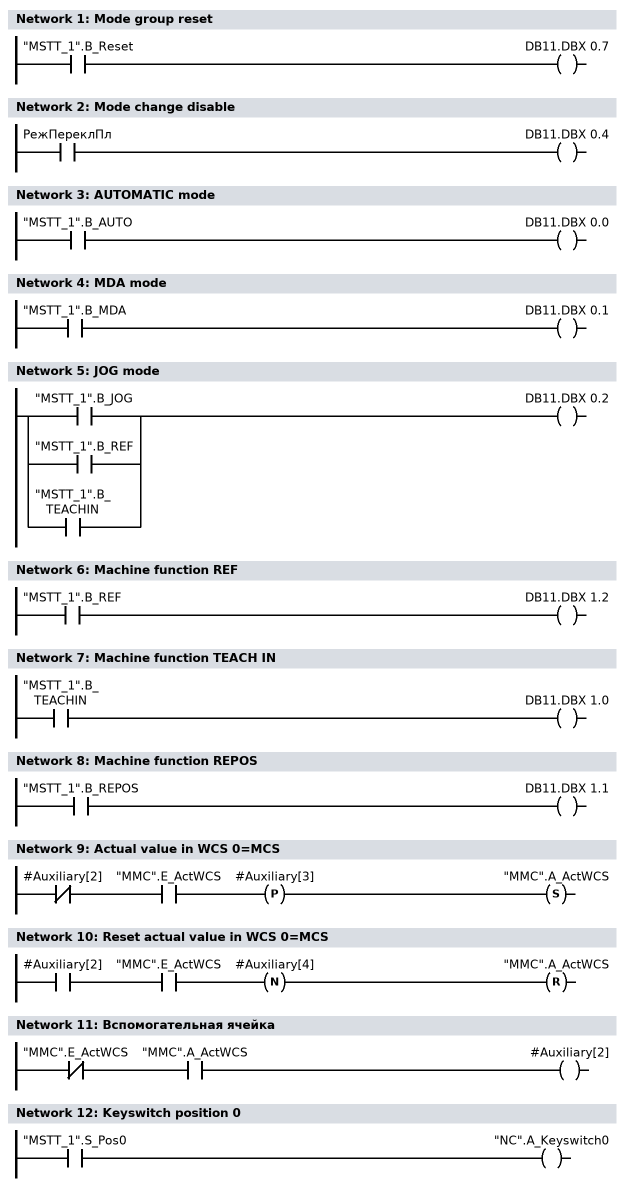
[picture p24: Lathe_Modes networks 1-12]
NETWORK
TITLE = Mode group reset
      A     "MSTT_1".B_Reset;
      =     DB11.DBX 0.7;
NETWORK
TITLE = Mode change disable 
      A     "РежПереклПл";
      =     DB11.DBX 0.4;
NETWORK
TITLE = AUTOMATIC mode
      A     "MSTT_1".B_AUTO;
      =     DB11.DBX 0.0;
NETWORK
TITLE = MDA mode
      A     "MSTT_1".B_MDA;
      =     DB11.DBX 0.1;
NETWORK
TITLE = JOG mode
      O     "MSTT_1".B_JOG;
      O     "MSTT_1".B_REF;
      O     "MSTT_1".B_TEACHIN;
      =     DB11.DBX 0.2;
NETWORK
TITLE = Machine function REF
      A     "MSTT_1".B_REF;
      =     DB11.DBX 1.2;
NETWORK
TITLE = Machine function TEACH IN
      A     "MSTT_1".B_TEACHIN;
      =     DB11.DBX 1.0;
NETWORK
TITLE = Machine function REPOS
      A     "MSTT_1".B_REPOS;
      =     DB11.DBX 1.1;
NETWORK
TITLE = Actual value in WCS 0=MCS
      AN    #Auxiliary[2];
      A     "MMC".E_ActWCS;
      FP    #Auxiliary[3];
      S     "MMC".A_ActWCS;
NETWORK
TITLE = Reset actual value in WCS 0=MCS
      A     #Auxiliary[2];
      A     "MMC".E_ActWCS;
      FN    #Auxiliary[4];
      R     "MMC".A_ActWCS;
NETWORK
TITLE = Вспомогательная ячейка
      AN    "MMC".E_ActWCS;
      A     "MMC".A_ActWCS;
      =     #Auxiliary[2];
NETWORK
TITLE = Keyswitch position 0
      A     "MSTT_1".S_Pos0;
      =     "NC".A_Keyswitch0;
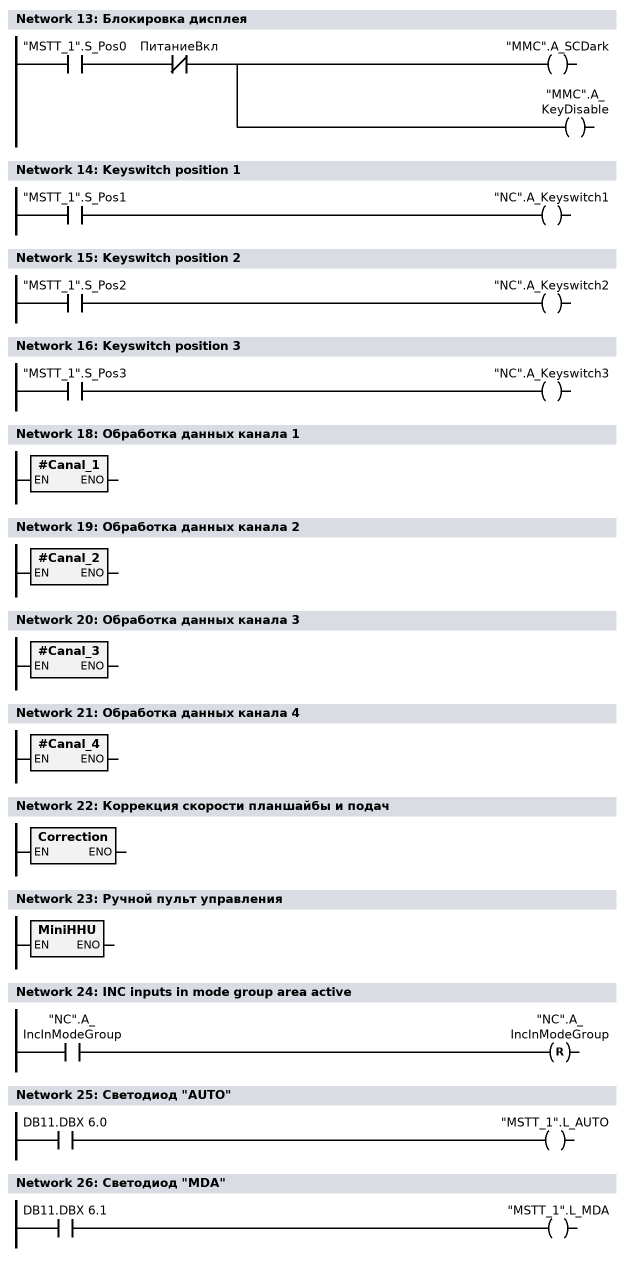
NETWORK
TITLE = Блокировка дисплея
      A     "MSTT_1".S_Pos0;
      AN    "ПитаниеВкл";
      =     "MMC".A_SCDark;
      =     "MMC".A_KeyDisable;
NETWORK
TITLE = Keyswitch position 1
      A     "MSTT_1".S_Pos1;
      =     "NC".A_Keyswitch1;
NETWORK
TITLE = Keyswitch position 2
      A     "MSTT_1".S_Pos2;
      =     "NC".A_Keyswitch2;
NETWORK
TITLE = Keyswitch position 3
      A     "MSTT_1".S_Pos3;
      =     "NC".A_Keyswitch3;
NETWORK
TITLE = Обработка вспомогательных функций
//      CALL  FC   107
      NOP   0;
NETWORK
TITLE = Обработка данных канала 1
      CALL  #Canal_1;
      NOP   0;
NETWORK
TITLE = Обработка данных канала 2
      CALL  #Canal_2;
      NOP   0;
NETWORK
TITLE = Обработка данных канала 3
      CALL  #Canal_3;
      NOP   0;
NETWORK
TITLE = Обработка данных канала 4
      CALL  #Canal_4;
      NOP   0;
NETWORK
TITLE = Коррекция скорости планшайбы и подач
      CALL  "Correction";
      NOP   0;
NETWORK
TITLE = Ручной пульт управления
      CALL  "MiniHHU";
      NOP   0;
NETWORK
TITLE = INC inputs in mode group area active
      A     "NC".A_IncInModeGroup;
      R     "NC".A_IncInModeGroup;
NETWORK
TITLE = Светодиод "AUTO"
      A     DB11.DBX 6.0;
      =     "MSTT_1".L_AUTO;
NETWORK
TITLE = Светодиод "MDA"
      A     DB11.DBX 6.1;
      =     "MSTT_1".L_MDA;
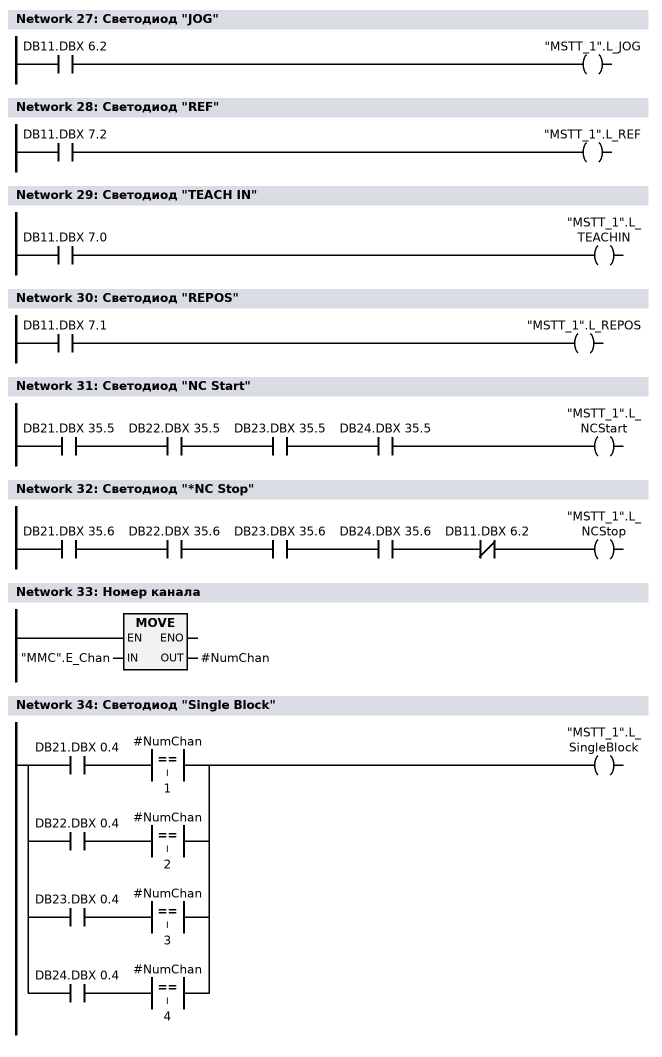
NETWORK
TITLE = Светодиод "JOG"
      A     DB11.DBX 6.2;
      =     "MSTT_1".L_JOG;
NETWORK
TITLE = Светодиод "REF"
      A     DB11.DBX 7.2;
      =     "MSTT_1".L_REF;
NETWORK
TITLE = Светодиод "TEACH IN"
      A     DB11.DBX 7.0;
      =     "MSTT_1".L_TEACHIN;
NETWORK
TITLE = Светодиод "REPOS"
      A     DB11.DBX 7.1;
      =     "MSTT_1".L_REPOS;
NETWORK
TITLE = Светодиод "NC Start"
      A     DB21.DBX 35.5;
      A     DB22.DBX 35.5;
      A     DB23.DBX 35.5;
      A     DB24.DBX 35.5;
      =     "MSTT_1".L_NCStart;
NETWORK
TITLE = Светодиод "*NC Stop"
      A     DB21.DBX 35.6;
      A     DB22.DBX 35.6;
      A     DB23.DBX 35.6;
      A     DB24.DBX 35.6;
      AN    DB11.DBX 6.2;
      =     "MSTT_1".L_NCStop;
NETWORK
TITLE = Номер канала
      L     "MMC".E_Chan;
      T     #NumChan;
      NOP   0;
NETWORK
TITLE = Светодиод "Single Block"
      A     DB21.DBX 0.4;
      A(;
      L     #NumChan;
      L     1;
      ==I;
      );
      O;
      A     DB22.DBX 0.4;
      A(;
      L     #NumChan;
      L     2;
      ==I;
      );
      O;
      A     DB23.DBX 0.4;
      A(;
      L     #NumChan;
      L     3;
      ==I;
      );
      O;
      A     DB24.DBX 0.4;
      A(;
      L     #NumChan;
      L     4;
      ==I;
      );
      =     "MSTT_1".L_SingleBlock;
END_FUNCTION_BLOCK

FUNCTION_BLOCK "Channel1_Modes"	// FB 106
AUTHOR : SEDIN
VERSION : 0.1
VAR
  Auxiliary : ARRAY  [0 .. 15 ] OF //Вспомогательная ячейка
  BOOL ;
  Table : FB 100;
  Support : FB 101;
END_VAR
VAR_TEMP
  NumChan : INT ;	//Номер канала
  B_SingleBlock : BOOL ;	//Клавиша SingleBlock
END_VAR
BEGIN
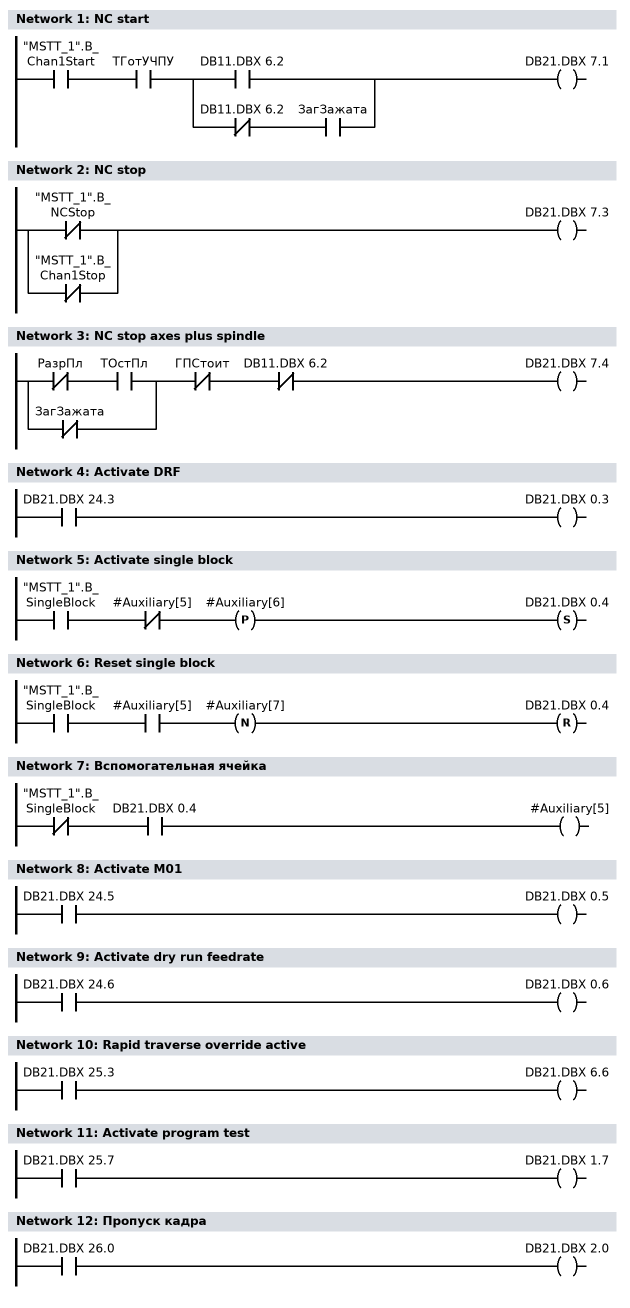
NETWORK
TITLE = NC start
      A     "MSTT_1".B_Chan1Start;
      A     "ТГотУЧПУ";
      A(;
      O     DB11.DBX 6.2;
      O;
      AN    DB11.DBX 6.2;
      A     "ЗагЗажата";
      );
      =     DB21.DBX 7.1;
NETWORK
TITLE = NC stop
      ON    "MSTT_1".B_NCStop;
      ON    "MSTT_1".B_Chan1Stop;
      =     DB21.DBX 7.3;
NETWORK
TITLE = NC stop axes plus spindle
      A(;
      AN    "РазрПл";
      A     "ТОстПл";
      ON    "ЗагЗажата";
      );
      AN    "ГПСтоит";
      AN    DB11.DBX 6.2;
      =     DB21.DBX 7.4;
NETWORK
TITLE = Activate DRF
      A     DB21.DBX 24.3;
      =     DB21.DBX 0.3;
NETWORK
TITLE = Activate single block
      A     "MSTT_1".B_SingleBlock;
      AN    #Auxiliary[5];
      FP    #Auxiliary[6];
      S     DB21.DBX 0.4;
NETWORK
TITLE = Reset single block
      A     "MSTT_1".B_SingleBlock;
      A     #Auxiliary[5];
      FN    #Auxiliary[7];
      R     DB21.DBX 0.4;
NETWORK
TITLE = Вспомогательная ячейка
      AN    "MSTT_1".B_SingleBlock;
      A     DB21.DBX 0.4;
      =     #Auxiliary[5];
NETWORK
TITLE = Activate M01
      A     DB21.DBX 24.5;
      =     DB21.DBX 0.5;
NETWORK
TITLE = Activate dry run feedrate
      A     DB21.DBX 24.6;
      =     DB21.DBX 0.6;
NETWORK
TITLE = Rapid traverse override active
      A     DB21.DBX 25.3;
      =     DB21.DBX 6.6;
NETWORK
TITLE = Activate program test
      A     DB21.DBX 25.7;
      =     DB21.DBX 1.7;
NETWORK
TITLE = Пропуск кадра
      A     DB21.DBX 26.0;
      =     DB21.DBX 2.0;
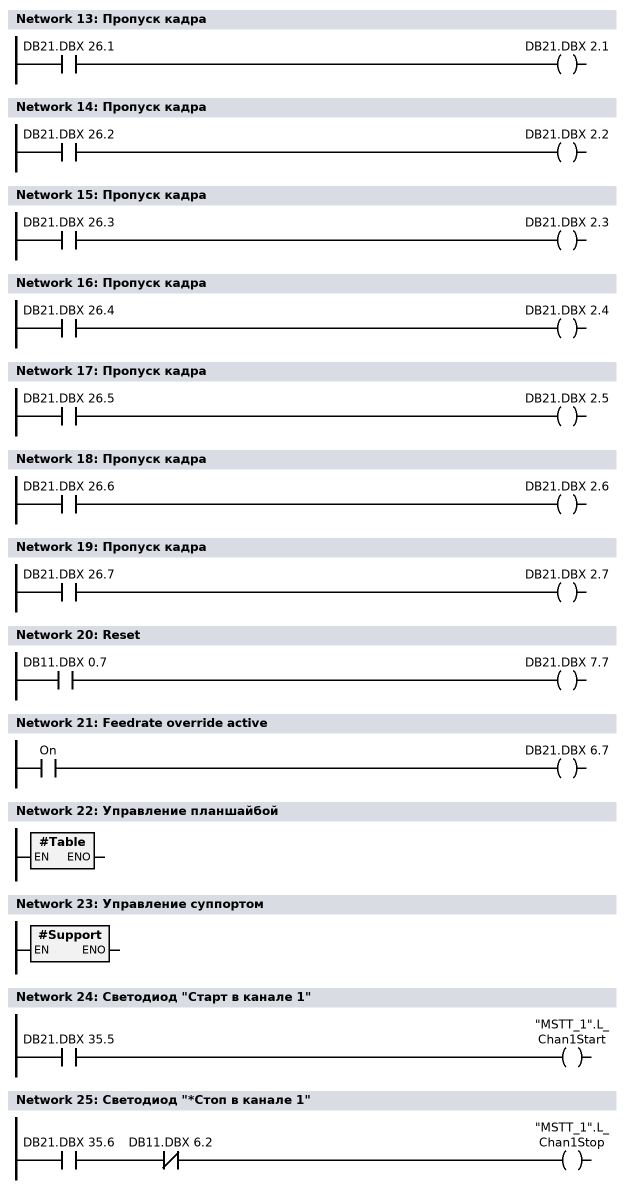
NETWORK
TITLE = Пропуск кадра
      A     DB21.DBX 26.1;
      =     DB21.DBX 2.1;
NETWORK
TITLE = Пропуск кадра
      A     DB21.DBX 26.2;
      =     DB21.DBX 2.2;
NETWORK
TITLE = Пропуск кадра
      A     DB21.DBX 26.3;
      =     DB21.DBX 2.3;
NETWORK
TITLE = Пропуск кадра
      A     DB21.DBX 26.4;
      =     DB21.DBX 2.4;
NETWORK
TITLE = Пропуск кадра
      A     DB21.DBX 26.5;
      =     DB21.DBX 2.5;
NETWORK
TITLE = Пропуск кадра
      A     DB21.DBX 26.6;
      =     DB21.DBX 2.6;
NETWORK
TITLE = Пропуск кадра
      A     DB21.DBX 26.7;
      =     DB21.DBX 2.7;
NETWORK
TITLE = Reset
      A     DB11.DBX 0.7;
      =     DB21.DBX 7.7;
NETWORK
TITLE = Feedrate override active
      A     "On";
      =     DB21.DBX 6.7;
NETWORK
TITLE = Управление планшайбой
      CALL  #Table;
      NOP   0;
NETWORK
TITLE = Управление суппортом
      CALL  #Support;
      NOP   0;
NETWORK
TITLE = Светодиод "Старт в канале 1"
      A     DB21.DBX 35.5;
      =     "MSTT_1".L_Chan1Start;
NETWORK
TITLE = Светодиод "*Стоп в канале 1"
      A     DB21.DBX 35.6;
      AN    DB11.DBX 6.2;
      =     "MSTT_1".L_Chan1Stop;
END_FUNCTION_BLOCK

FUNCTION_BLOCK "Channel2_Modes"	// FB 107
AUTHOR : SEDIN
VERSION : 0.1
VAR
  Auxiliary : ARRAY  [0 .. 15 ] OF //Вспомогательная ячейка
  BOOL ;
  Support : FB 102;
END_VAR
VAR_TEMP
  NumChan : INT ;	//Номер канала
  B_SingleBlock : BOOL ;	//Клавиша SingleBlock
END_VAR
BEGIN
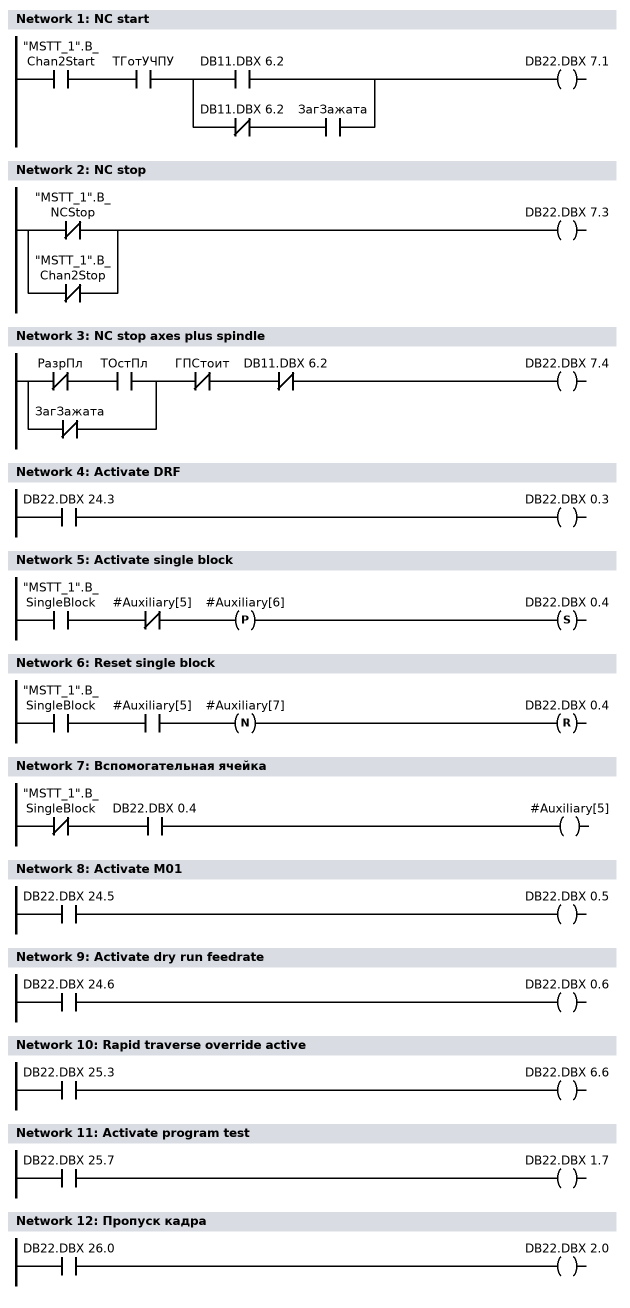
NETWORK
TITLE = NC start
      A     "MSTT_1".B_Chan2Start;
      A     "ТГотУЧПУ";
      A(;
      O     DB11.DBX 6.2;
      O;
      AN    DB11.DBX 6.2;
      A     "ЗагЗажата";
      );
      =     DB22.DBX 7.1;
NETWORK
TITLE = NC stop
      ON    "MSTT_1".B_NCStop;
      ON    "MSTT_1".B_Chan2Stop;
      =     DB22.DBX 7.3;
NETWORK
TITLE = NC stop axes plus spindle
      A(;
      AN    "РазрПл";
      A     "ТОстПл";
      ON    "ЗагЗажата";
      );
      AN    "ГПСтоит";
      AN    DB11.DBX 6.2;
      =     DB22.DBX 7.4;
NETWORK
TITLE = Activate DRF
      A     DB22.DBX 24.3;
      =     DB22.DBX 0.3;
NETWORK
TITLE = Activate single block
      A     "MSTT_1".B_SingleBlock;
      AN    #Auxiliary[5];
      FP    #Auxiliary[6];
      S     DB22.DBX 0.4;
NETWORK
TITLE = Reset single block
      A     "MSTT_1".B_SingleBlock;
      A     #Auxiliary[5];
      FN    #Auxiliary[7];
      R     DB22.DBX 0.4;
NETWORK
TITLE = Вспомогательная ячейка
      AN    "MSTT_1".B_SingleBlock;
      A     DB22.DBX 0.4;
      =     #Auxiliary[5];
NETWORK
TITLE = Activate M01
      A     DB22.DBX 24.5;
      =     DB22.DBX 0.5;
NETWORK
TITLE = Activate dry run feedrate
      A     DB22.DBX 24.6;
      =     DB22.DBX 0.6;
NETWORK
TITLE = Rapid traverse override active
      A     DB22.DBX 25.3;
      =     DB22.DBX 6.6;
NETWORK
TITLE = Activate program test
      A     DB22.DBX 25.7;
      =     DB22.DBX 1.7;
NETWORK
TITLE = Пропуск кадра
      A     DB22.DBX 26.0;
      =     DB22.DBX 2.0;
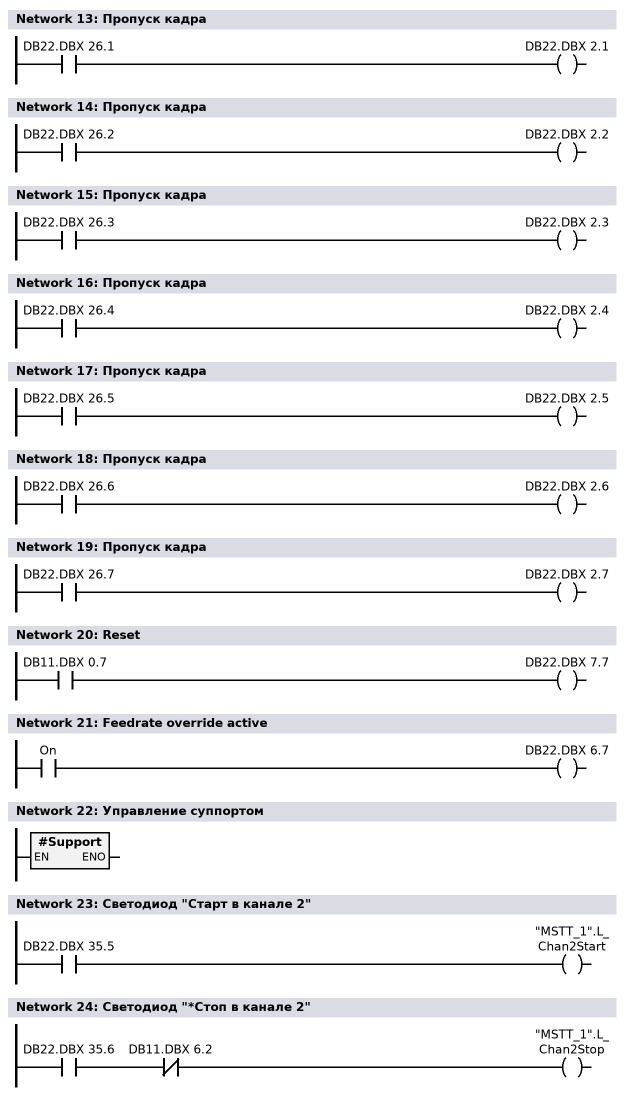
NETWORK
TITLE = Пропуск кадра
      A     DB22.DBX 26.1;
      =     DB22.DBX 2.1;
NETWORK
TITLE = Пропуск кадра
      A     DB22.DBX 26.2;
      =     DB22.DBX 2.2;
NETWORK
TITLE = Пропуск кадра
      A     DB22.DBX 26.3;
      =     DB22.DBX 2.3;
NETWORK
TITLE = Пропуск кадра
      A     DB22.DBX 26.4;
      =     DB22.DBX 2.4;
NETWORK
TITLE = Пропуск кадра
      A     DB22.DBX 26.5;
      =     DB22.DBX 2.5;
NETWORK
TITLE = Пропуск кадра
      A     DB22.DBX 26.6;
      =     DB22.DBX 2.6;
NETWORK
TITLE = Пропуск кадра
      A     DB22.DBX 26.7;
      =     DB22.DBX 2.7;
NETWORK
TITLE = Reset
      A     DB11.DBX 0.7;
      =     DB22.DBX 7.7;
NETWORK
TITLE = Feedrate override active
      A     "On";
      =     DB22.DBX 6.7;
NETWORK
TITLE = Управление суппортом
      CALL  #Support;
      NOP   0;
NETWORK
TITLE = Светодиод "Старт в канале 2"
      A     DB22.DBX 35.5;
      =     "MSTT_1".L_Chan2Start;
NETWORK
TITLE = Светодиод "*Стоп в канале 2"
      A     DB22.DBX 35.6;
      AN    DB11.DBX 6.2;
      =     "MSTT_1".L_Chan2Stop;
END_FUNCTION_BLOCK

FUNCTION_BLOCK "Channel3_Modes"	// FB 108
AUTHOR : SEDIN
VERSION : 0.1
VAR
  Auxiliary : ARRAY  [0 .. 15 ] OF //Вспомогательная ячейка
  BOOL ;
  Support : FB 103;
END_VAR
VAR_TEMP
  NumChan : INT ;	//Номер канала
  B_SingleBlock : BOOL ;	//Клавиша SingleBlock
END_VAR
BEGIN
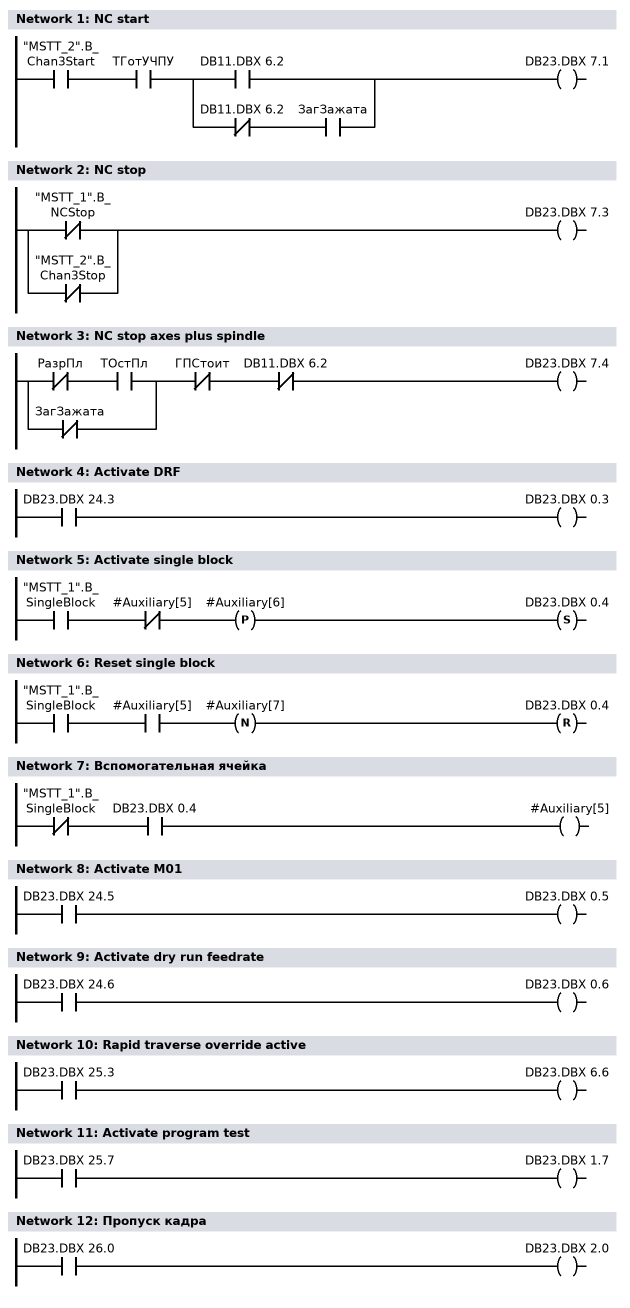
NETWORK
TITLE = NC start
      A     "MSTT_2".B_Chan3Start;
      A     "ТГотУЧПУ";
      A(;
      O     DB11.DBX 6.2;
      O;
      AN    DB11.DBX 6.2;
      A     "ЗагЗажата";
      );
      =     DB23.DBX 7.1;
NETWORK
TITLE = NC stop
      ON    "MSTT_1".B_NCStop;
      ON    "MSTT_2".B_Chan3Stop;
      =     DB23.DBX 7.3;
NETWORK
TITLE = NC stop axes plus spindle
      A(;
      AN    "РазрПл";
      A     "ТОстПл";
      ON    "ЗагЗажата";
      );
      AN    "ГПСтоит";
      AN    DB11.DBX 6.2;
      =     DB23.DBX 7.4;
NETWORK
TITLE = Activate DRF
      A     DB23.DBX 24.3;
      =     DB23.DBX 0.3;
NETWORK
TITLE = Activate single block
      A     "MSTT_1".B_SingleBlock;
      AN    #Auxiliary[5];
      FP    #Auxiliary[6];
      S     DB23.DBX 0.4;
NETWORK
TITLE = Reset single block
      A     "MSTT_1".B_SingleBlock;
      A     #Auxiliary[5];
      FN    #Auxiliary[7];
      R     DB23.DBX 0.4;
NETWORK
TITLE = Вспомогательная ячейка
      AN    "MSTT_1".B_SingleBlock;
      A     DB23.DBX 0.4;
      =     #Auxiliary[5];
NETWORK
TITLE = Activate M01
      A     DB23.DBX 24.5;
      =     DB23.DBX 0.5;
NETWORK
TITLE = Activate dry run feedrate
      A     DB23.DBX 24.6;
      =     DB23.DBX 0.6;
NETWORK
TITLE = Rapid traverse override active
      A     DB23.DBX 25.3;
      =     DB23.DBX 6.6;
NETWORK
TITLE = Activate program test
      A     DB23.DBX 25.7;
      =     DB23.DBX 1.7;
NETWORK
TITLE = Пропуск кадра
      A     DB23.DBX 26.0;
      =     DB23.DBX 2.0;
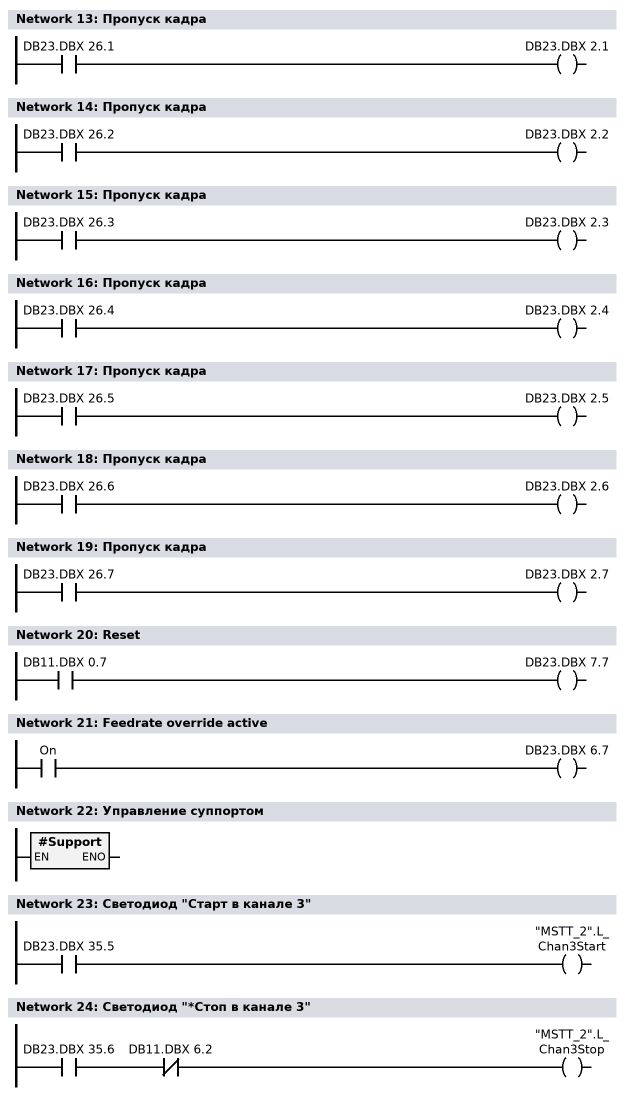
NETWORK
TITLE = Пропуск кадра
      A     DB23.DBX 26.1;
      =     DB23.DBX 2.1;
NETWORK
TITLE = Пропуск кадра
      A     DB23.DBX 26.2;
      =     DB23.DBX 2.2;
NETWORK
TITLE = Пропуск кадра
      A     DB23.DBX 26.3;
      =     DB23.DBX 2.3;
NETWORK
TITLE = Пропуск кадра
      A     DB23.DBX 26.4;
      =     DB23.DBX 2.4;
NETWORK
TITLE = Пропуск кадра
      A     DB23.DBX 26.5;
      =     DB23.DBX 2.5;
NETWORK
TITLE = Пропуск кадра
      A     DB23.DBX 26.6;
      =     DB23.DBX 2.6;
NETWORK
TITLE = Пропуск кадра
      A     DB23.DBX 26.7;
      =     DB23.DBX 2.7;
NETWORK
TITLE = Reset
      A     DB11.DBX 0.7;
      =     DB23.DBX 7.7;
NETWORK
TITLE = Feedrate override active
      A     "On";
      =     DB23.DBX 6.7;
NETWORK
TITLE = Управление суппортом
      CALL  #Support;
      NOP   0;
NETWORK
TITLE = Светодиод "Старт в канале 3"
      A     DB23.DBX 35.5;
      =     "MSTT_2".L_Chan3Start;
NETWORK
TITLE = Светодиод "*Стоп в канале 3"
      A     DB23.DBX 35.6;
      AN    DB11.DBX 6.2;
      =     "MSTT_2".L_Chan3Stop;
END_FUNCTION_BLOCK

FUNCTION_BLOCK "Channel4_Modes"	// FB 109
AUTHOR : SEDIN
VERSION : 0.1
VAR
  Auxiliary : ARRAY  [0 .. 15 ] OF //Вспомогательная ячейка
  BOOL ;
  Support : FB 104;
END_VAR
VAR_TEMP
  NumChan : INT ;	//Номер канала
  B_SingleBlock : BOOL ;	//Клавиша SingleBlock
END_VAR
BEGIN
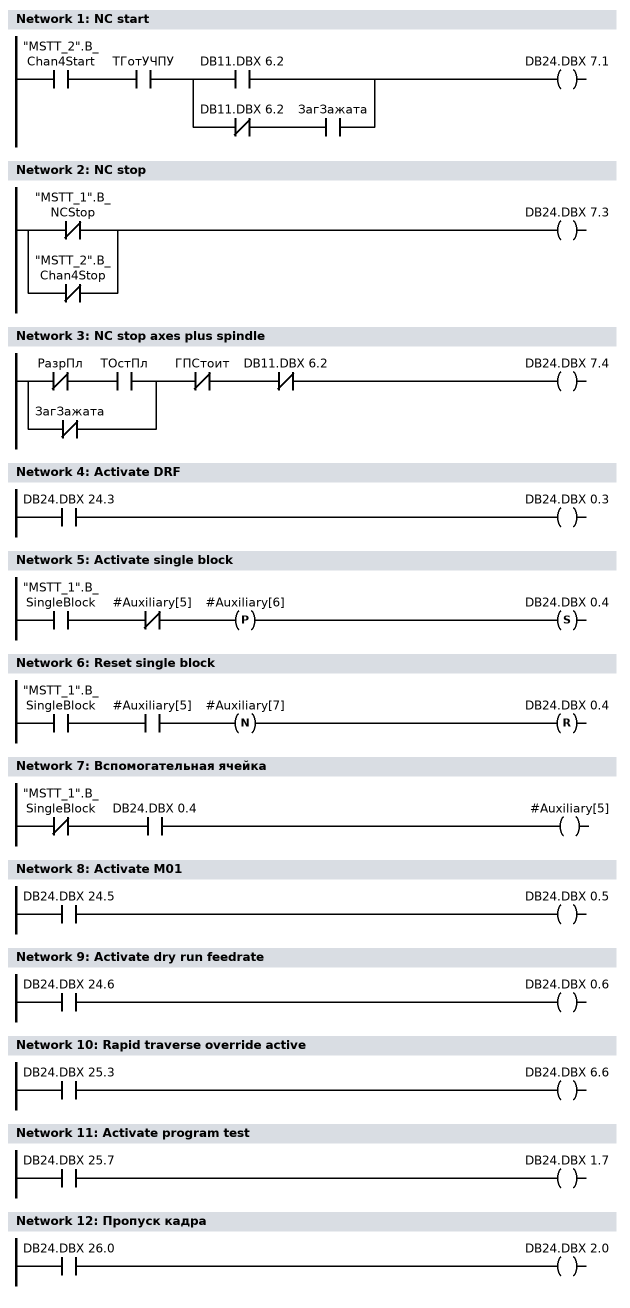
NETWORK
TITLE = NC start
      A     "MSTT_2".B_Chan4Start;
      A     "ТГотУЧПУ";
      A(;
      O     DB11.DBX 6.2;
      O;
      AN    DB11.DBX 6.2;
      A     "ЗагЗажата";
      );
      =     DB24.DBX 7.1;
NETWORK
TITLE = NC stop
      ON    "MSTT_1".B_NCStop;
      ON    "MSTT_2".B_Chan4Stop;
      =     DB24.DBX 7.3;
NETWORK
TITLE = NC stop axes plus spindle
      A(;
      AN    "РазрПл";
      A     "ТОстПл";
      ON    "ЗагЗажата";
      );
      AN    "ГПСтоит";
      AN    DB11.DBX 6.2;
      =     DB24.DBX 7.4;
NETWORK
TITLE = Activate DRF
      A     DB24.DBX 24.3;
      =     DB24.DBX 0.3;
NETWORK
TITLE = Activate single block
      A     "MSTT_1".B_SingleBlock;
      AN    #Auxiliary[5];
      FP    #Auxiliary[6];
      S     DB24.DBX 0.4;
NETWORK
TITLE = Reset single block
      A     "MSTT_1".B_SingleBlock;
      A     #Auxiliary[5];
      FN    #Auxiliary[7];
      R     DB24.DBX 0.4;
NETWORK
TITLE = Вспомогательная ячейка
      AN    "MSTT_1".B_SingleBlock;
      A     DB24.DBX 0.4;
      =     #Auxiliary[5];
NETWORK
TITLE = Activate M01
      A     DB24.DBX 24.5;
      =     DB24.DBX 0.5;
NETWORK
TITLE = Activate dry run feedrate
      A     DB24.DBX 24.6;
      =     DB24.DBX 0.6;
NETWORK
TITLE = Rapid traverse override active
      A     DB24.DBX 25.3;
      =     DB24.DBX 6.6;
NETWORK
TITLE = Activate program test
      A     DB24.DBX 25.7;
      =     DB24.DBX 1.7;
NETWORK
TITLE = Пропуск кадра
      A     DB24.DBX 26.0;
      =     DB24.DBX 2.0;
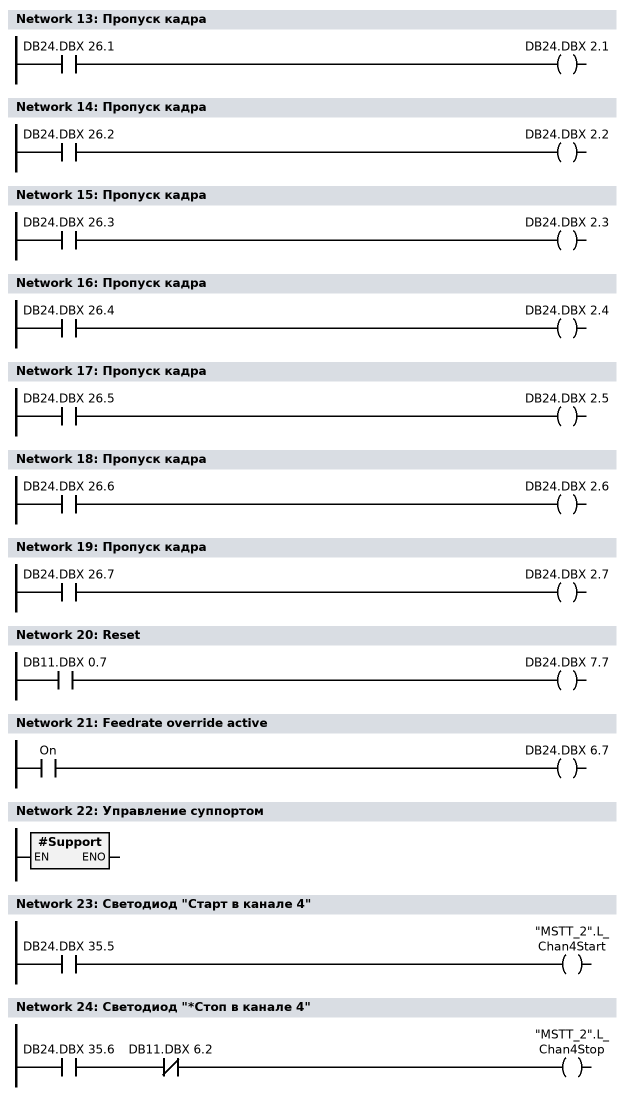
NETWORK
TITLE = Пропуск кадра
      A     DB24.DBX 26.1;
      =     DB24.DBX 2.1;
NETWORK
TITLE = Пропуск кадра
      A     DB24.DBX 26.2;
      =     DB24.DBX 2.2;
NETWORK
TITLE = Пропуск кадра
      A     DB24.DBX 26.3;
      =     DB24.DBX 2.3;
NETWORK
TITLE = Пропуск кадра
      A     DB24.DBX 26.4;
      =     DB24.DBX 2.4;
NETWORK
TITLE = Пропуск кадра
      A     DB24.DBX 26.5;
      =     DB24.DBX 2.5;
NETWORK
TITLE = Пропуск кадра
      A     DB24.DBX 26.6;
      =     DB24.DBX 2.6;
NETWORK
TITLE = Пропуск кадра
      A     DB24.DBX 26.7;
      =     DB24.DBX 2.7;
NETWORK
TITLE = Reset
      A     DB11.DBX 0.7;
      =     DB24.DBX 7.7;
NETWORK
TITLE = Feedrate override active
      A     "On";
      =     DB24.DBX 6.7;
NETWORK
TITLE = Управление суппортом
      CALL  #Support;
      NOP   0;
NETWORK
TITLE = Светодиод "Старт в канале 4"
      A     DB24.DBX 35.5;
      =     "MSTT_2".L_Chan4Start;
NETWORK
TITLE = Светодиод "*Стоп в канале 4"
      A     DB24.DBX 35.6;
      AN    DB11.DBX 6.2;
      =     "MSTT_2".L_Chan4Stop;
END_FUNCTION_BLOCK

FUNCTION_BLOCK "Support_Lub"	// FB 121
AUTHOR : SEDIN
VERSION : 0.1
VAR_INPUT
  Permission : BOOL ;	//Разрешение работы насоса ИСС
  LubButton : BOOL ;	//Кнопка принудительной прокачки ИСС
  Pressure : BOOL ;	//Реле давления ИСС
  Level : BOOL ;	//Реле уровня ИСС
  BlockError : BOOL ;	//Блокировка ошибки смазки
END_VAR
VAR_OUTPUT
  Pump : BOOL ;	//Команда на смазку суппорта
  LubError : BOOL ;	//Ошибка смазки суппорта
  Message1 : BOOL ;	//Сообщение о низком уровне масла
  Message2 : BOOL ;	//Сообщение об отсутствии набора давления
  Message3 : BOOL ;	//Сообщение об отсутствии падения давления
END_VAR
VAR
  Mem_1 : BOOL ;	//Память фронта сигнала 1
  Mem_2 : BOOL ;	//Память фронта сигнала 2
  ResetTimers : BOOL ;	//Сброс таймеров смазки суппорта
  TLubError_In : BOOL ;	//Пуск таймера задержки реакции на ошибку смазки
  TLubInterval_In : BOOL ;	//Пуск таймера интервала прокачки ИСС
  TLubDelay_In : BOOL ;	//Пуск таймера задержки на прокачку ИСС
  TLubError_Q : BOOL ;	//Таймер задержки реакции на ошибку смазки сработал
  TLubInterval_Q : BOOL ;	//Таймер интервала прокачки ИСС сработал
  TLubDelay_Q : BOOL ;	//Таймер задержки на прокачку ИСС сработал
  TLubError : SFB 4;	//Задержка реакции на ошибку смазки
  TLubInterval : SFB 4;	//Таймер интервала прокачки ИСС
  TLubDelay : SFB 4;	//Задержка на прокачку ИСС
END_VAR
BEGIN
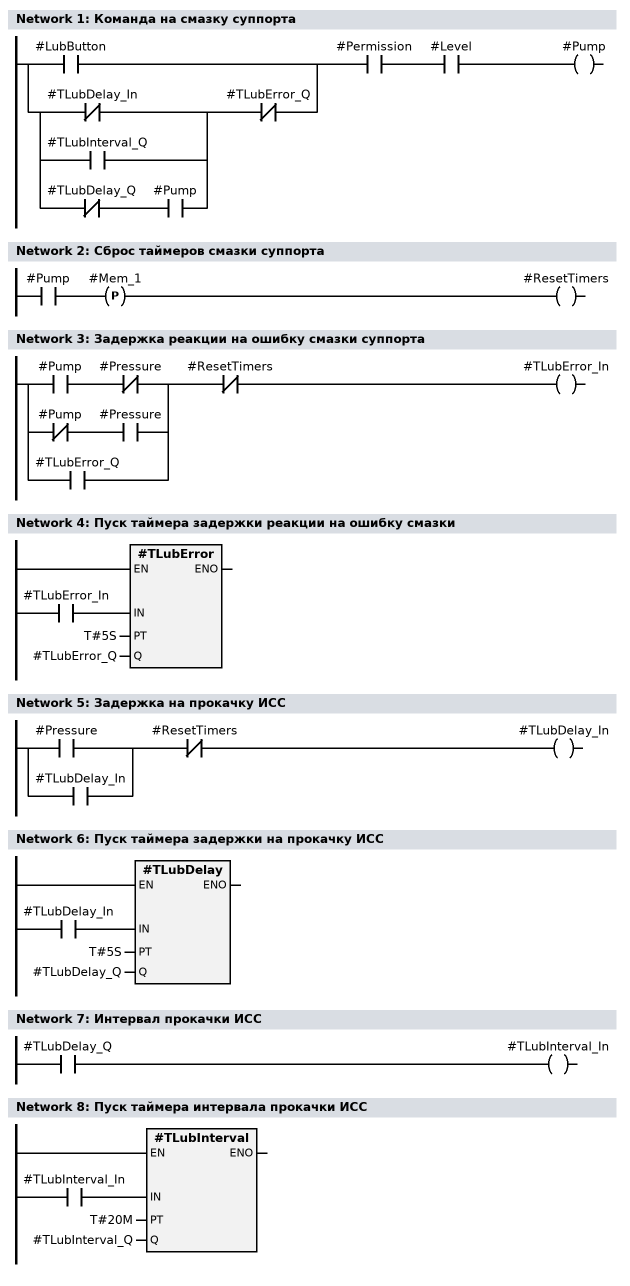
NETWORK
TITLE = Команда на смазку суппорта
      A(;
      O     #LubButton;
      O;
      A(;
      ON    #TLubDelay_In;
      O     #TLubInterval_Q;
      O;
      AN    #TLubDelay_Q;
      A     #Pump;
      );
      AN    #TLubError_Q;
      );
      A     #Permission;
      A     #Level;
      =     #Pump;
NETWORK
TITLE = Сброс таймеров смазки суппорта
      A     #Pump;
      FP    #Mem_1;
      =     #ResetTimers;
NETWORK
TITLE = Задержка реакции на ошибку смазки суппорта
      A(;
      A     #Pump;
      AN    #Pressure;
      O;
      AN    #Pump;
      A     #Pressure;
      O     #TLubError_Q;
      );
      AN    #ResetTimers;
      =     #TLubError_In;
NETWORK
TITLE = Пуск таймера задержки реакции на ошибку смазки
      A     #TLubError_In;
      =     L 0.0;
      BLD   103;
      CALL  #TLubError (
           IN                       := L 0.0,
           PT                       := T#5S,
           Q                        := #TLubError_Q);
      NOP   0;
NETWORK
TITLE = Задержка на прокачку ИСС
      A(;
      O     #Pressure;
      O     #TLubDelay_In;
      );
      AN    #ResetTimers;
      =     #TLubDelay_In;
NETWORK
TITLE = Пуск таймера задержки на прокачку ИСС 
      A     #TLubDelay_In;
      =     L 0.0;
      BLD   103;
      CALL  #TLubDelay (
           IN                       := L 0.0,
           PT                       := T#5S,
           Q                        := #TLubDelay_Q);
      NOP   0;
NETWORK
TITLE = Интервал прокачки ИСС
      A     #TLubDelay_Q;
      =     #TLubInterval_In;
NETWORK
TITLE = Пуск таймера интервала прокачки ИСС
      A     #TLubInterval_In;
      =     L 0.0;
      BLD   103;
      CALL  #TLubInterval (
           IN                       := L 0.0,
           PT                       := T#20M,
           Q                        := #TLubInterval_Q);
      NOP   0;
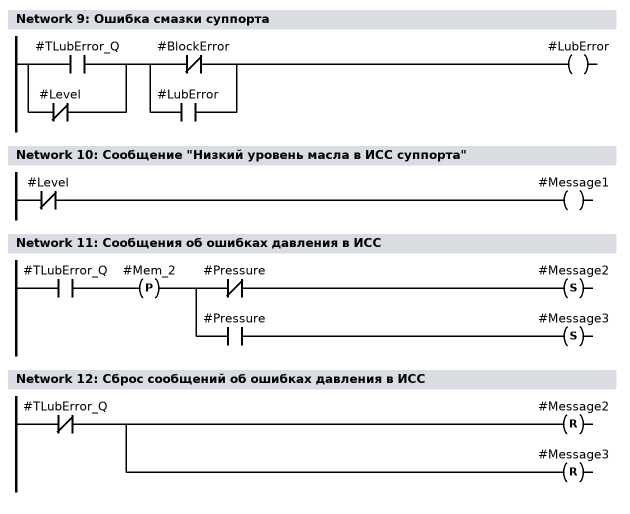
NETWORK
TITLE = Ошибка смазки суппорта
      A(;
      O     #TLubError_Q;
      ON    #Level;
      );
      A(;
      ON    #BlockError;
      O     #LubError;
      );
      =     #LubError;
NETWORK
TITLE = Сообщение "Низкий уровень масла в ИСС суппорта"
      AN    #Level;
      =     #Message1;
NETWORK
TITLE = Сообщения об ошибках давления в ИСС
      A     #TLubError_Q;
      FP    #Mem_2;
      =     L 0.0;
      A     L 0.0;
      AN    #Pressure;
      S     #Message2;
      A     L 0.0;
      A     #Pressure;
      S     #Message3;
NETWORK
TITLE = Сброс сообщений об ошибках давления в ИСС
      AN    #TLubError_Q;
      R     #Message2;
      R     #Message3;
END_FUNCTION_BLOCK

FUNCTION_BLOCK FB 1001
AUTHOR : SEDIN
VERSION : 0.1
VAR
  Auxiliary : ARRAY  [0 .. 15 ] OF //Вспомогательная ячейка
  BOOL ;
END_VAR
VAR_TEMP
  ActMoment : INT ;	//Текущий момент, ось 1
END_VAR
BEGIN
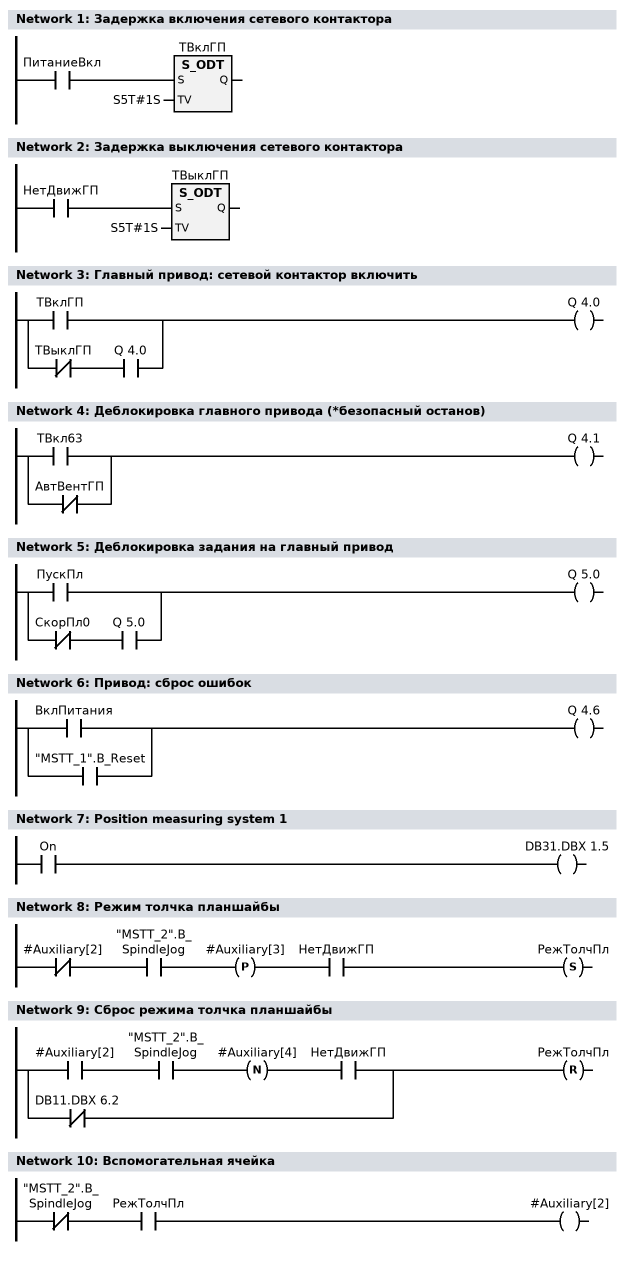
NETWORK
TITLE = Задержка включения сетевого контактора
      A     "ПитаниеВкл";
      L     S5T#1S;
      SD    "ТВклГП";
      NOP   0;
      NOP   0;
      NOP   0;
      NOP   0;
NETWORK
TITLE = Задержка выключения сетевого контактора
      A     "НетДвижГП";
      L     S5T#1S;
      SD    "ТВыклГП";
      NOP   0;
      NOP   0;
      NOP   0;
      NOP   0;
NETWORK
TITLE = Главный привод: сетевой контактор включить
      O     "ТВклГП";
      O;
      AN    "ТВыклГП";
      A     Q 4.0;
      =     Q 4.0;
NETWORK
TITLE = Деблокировка главного привода (*безопасный останов)
      O     "ТВкл63";
      ON    "АвтВентГП";
      =     Q 4.1;
NETWORK
TITLE = Деблокировка задания на главный привод
      O     "ПускПл";
      O;
      AN    "СкорПл0";
      A     Q 5.0;
      =     Q 5.0;
NETWORK
TITLE = Привод: сброс ошибок
      O     "ВклПитания";
      O     "MSTT_1".B_Reset;
      =     Q 4.6;
NETWORK
TITLE = Position measuring system 1
      A     "On";
      =     DB31.DBX 1.5;
NETWORK
TITLE = Режим толчка планшайбы
      AN    #Auxiliary[2];
      A     "MSTT_2".B_SpindleJog;
      FP    #Auxiliary[3];
      A     "НетДвижГП";
      S     "РежТолчПл";
NETWORK
TITLE = Сброс режима толчка планшайбы
      A     #Auxiliary[2];
      A     "MSTT_2".B_SpindleJog;
      FN    #Auxiliary[4];
      A     "НетДвижГП";
      ON    DB11.DBX 6.2;
      R     "РежТолчПл";
NETWORK
TITLE = Вспомогательная ячейка
      AN    "MSTT_2".B_SpindleJog;
      A     "РежТолчПл";
      =     #Auxiliary[2];
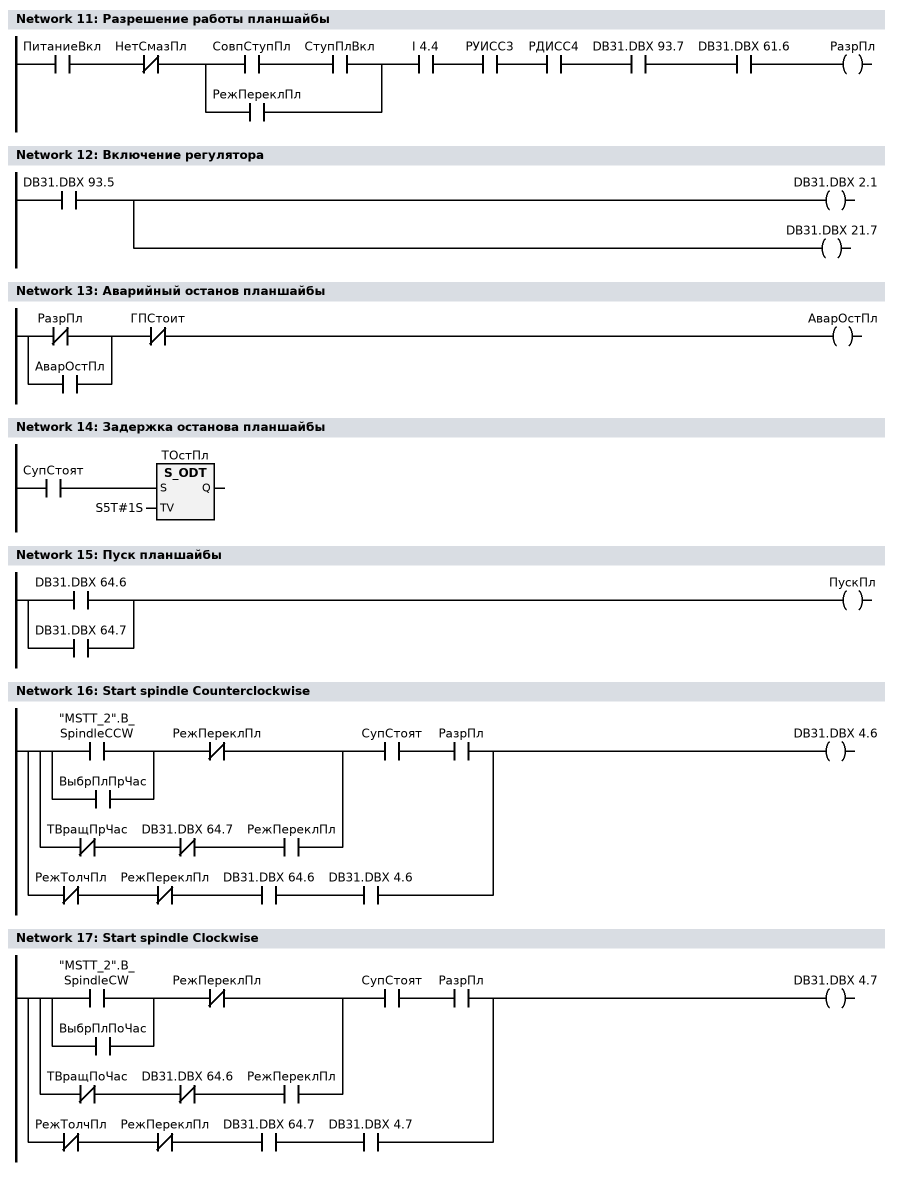
NETWORK
TITLE = Разрешение работы планшайбы
      A     "ПитаниеВкл";
      AN    "НетСмазПл";
      A(;
      A     "СовпСтупПл";
      A     "СтупПлВкл";
      O     "РежПереклПл";
      );
      A     I 4.4;
      A     "РУИСС3";
      A     "РДИСС4";
      A     DB31.DBX 93.7;
      A     DB31.DBX 61.6;
      =     "РазрПл";
NETWORK
TITLE = Включение регулятора
      A     DB31.DBX 93.5;
      =     DB31.DBX 2.1;
      =     DB31.DBX 21.7;
NETWORK
TITLE = Аварийный останов планшайбы
      A(;
      ON    "РазрПл";
      O     "АварОстПл";
      );
      AN    "ГПСтоит";
      =     "АварОстПл";
NETWORK
TITLE = Задержка останова планшайбы
      A     "СупСтоят";
      L     S5T#1S;
      SD    "ТОстПл";
      NOP   0;
      NOP   0;
      NOP   0;
      NOP   0;
NETWORK
TITLE = Пуск планшайбы
      O     DB31.DBX 64.6;
      O     DB31.DBX 64.7;
      =     "ПускПл";
NETWORK
TITLE = Start spindle Counterclockwise
      A(;
      A(;
      O     "MSTT_2".B_SpindleCCW;
      O     "ВыбрПлПрЧас";
      );
      AN    "РежПереклПл";
      O;
      AN    "ТВращПрЧас";
      AN    DB31.DBX 64.7;
      A     "РежПереклПл";
      );
      A     "СупСтоят";
      A     "РазрПл";
      O;
      AN    "РежТолчПл";
      AN    "РежПереклПл";
      A     DB31.DBX 64.6;
      A     DB31.DBX 4.6;
      =     DB31.DBX 4.6;
NETWORK
TITLE = Start spindle Clockwise
      A(;
      A(;
      O     "MSTT_2".B_SpindleCW;
      O     "ВыбрПлПоЧас";
      );
      AN    "РежПереклПл";
      O;
      AN    "ТВращПоЧас";
      AN    DB31.DBX 64.6;
      A     "РежПереклПл";
      );
      A     "СупСтоят";
      A     "РазрПл";
      O;
      AN    "РежТолчПл";
      AN    "РежПереклПл";
      A     DB31.DBX 64.7;
      A     DB31.DBX 4.7;
      =     DB31.DBX 4.7;
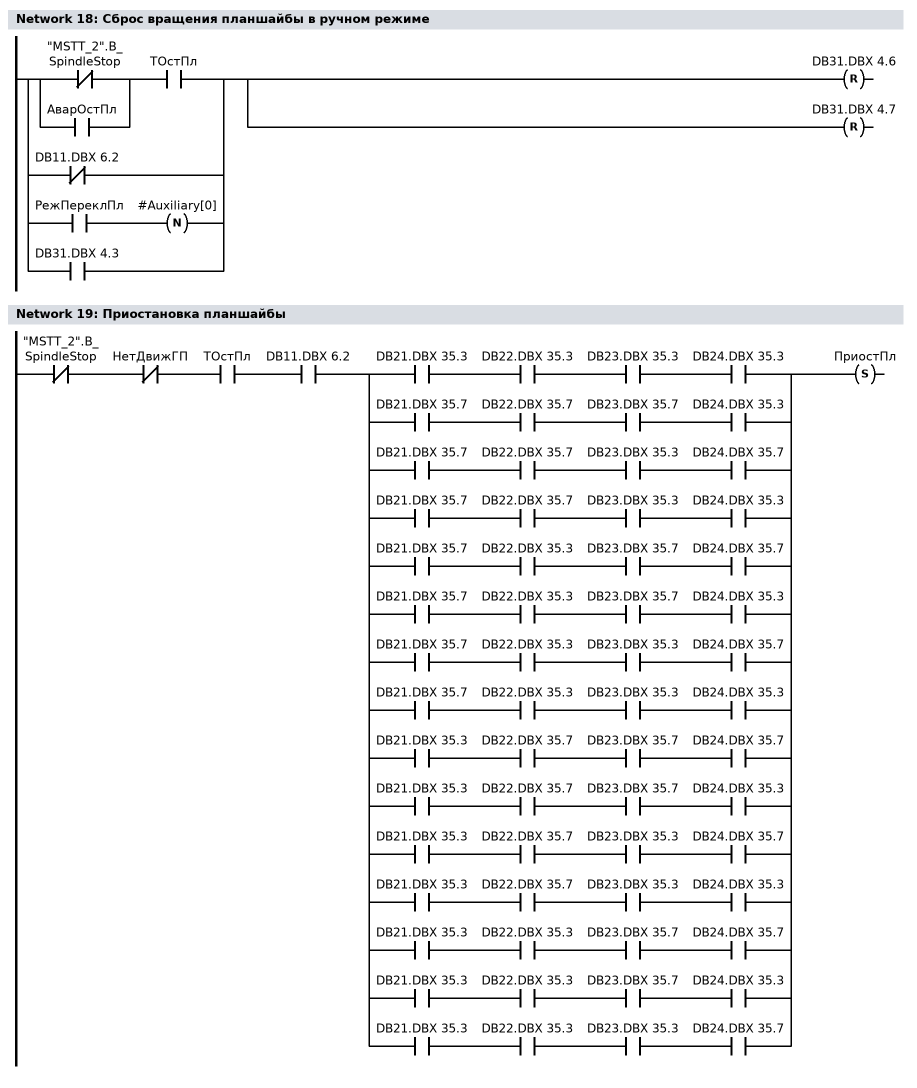
NETWORK
TITLE = Сброс вращения планшайбы в ручном режиме
      A(;
      ON    "MSTT_2".B_SpindleStop;
      O     "АварОстПл";
      );
      A     "ТОстПл";
      ON    DB11.DBX 6.2;
      O(;
      A     "РежПереклПл";
      BLD   100;
      FN    #Auxiliary[0];
      );
      O     DB31.DBX 4.3;
      R     DB31.DBX 4.6;
      R     DB31.DBX 4.7;
NETWORK
TITLE = Приостановка планшайбы
      AN    "MSTT_2".B_SpindleStop;
      AN    "НетДвижГП";
      A     "ТОстПл";
      A     DB11.DBX 6.2;
      A(;
      A     DB21.DBX 35.3;
      A     DB22.DBX 35.3;
      A     DB23.DBX 35.3;
      A     DB24.DBX 35.3;
      O;
      A     DB21.DBX 35.7;
      A     DB22.DBX 35.7;
      A     DB23.DBX 35.7;
      A     DB24.DBX 35.3;
      O;
      A     DB21.DBX 35.7;
      A     DB22.DBX 35.7;
      A     DB23.DBX 35.3;
      A     DB24.DBX 35.7;
      O;
      A     DB21.DBX 35.7;
      A     DB22.DBX 35.7;
      A     DB23.DBX 35.3;
      A     DB24.DBX 35.3;
      O;
      A     DB21.DBX 35.7;
      A     DB22.DBX 35.3;
      A     DB23.DBX 35.7;
      A     DB24.DBX 35.7;
      O;
      A     DB21.DBX 35.7;
      A     DB22.DBX 35.3;
      A     DB23.DBX 35.7;
      A     DB24.DBX 35.3;
      O;
      A     DB21.DBX 35.7;
      A     DB22.DBX 35.3;
      A     DB23.DBX 35.3;
      A     DB24.DBX 35.7;
      O;
      A     DB21.DBX 35.7;
      A     DB22.DBX 35.3;
      A     DB23.DBX 35.3;
      A     DB24.DBX 35.3;
      O;
      A     DB21.DBX 35.3;
      A     DB22.DBX 35.7;
      A     DB23.DBX 35.7;
      A     DB24.DBX 35.7;
      O;
      A     DB21.DBX 35.3;
      A     DB22.DBX 35.7;
      A     DB23.DBX 35.7;
      A     DB24.DBX 35.3;
      O;
      A     DB21.DBX 35.3;
      A     DB22.DBX 35.7;
      A     DB23.DBX 35.3;
      A     DB24.DBX 35.7;
      O;
      A     DB21.DBX 35.3;
      A     DB22.DBX 35.7;
      A     DB23.DBX 35.3;
      A     DB24.DBX 35.3;
      O;
      A     DB21.DBX 35.3;
      A     DB22.DBX 35.3;
      A     DB23.DBX 35.7;
      A     DB24.DBX 35.7;
      O;
      A     DB21.DBX 35.3;
      A     DB22.DBX 35.3;
      A     DB23.DBX 35.7;
      A     DB24.DBX 35.3;
      O;
      A     DB21.DBX 35.3;
      A     DB22.DBX 35.3;
      A     DB23.DBX 35.3;
      A     DB24.DBX 35.7;
      );
      S     "ПриостПл";
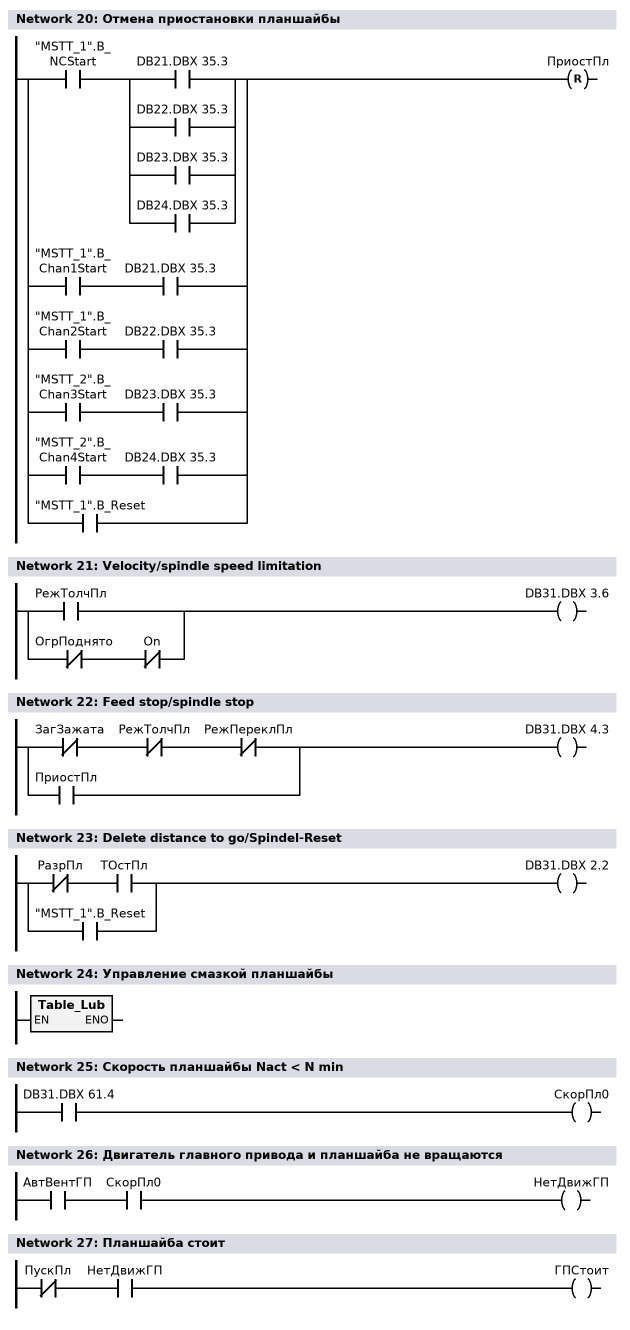
NETWORK
TITLE = Отмена приостановки планшайбы
      A     "MSTT_1".B_NCStart;
      A(;
      O     DB21.DBX 35.3;
      O     DB22.DBX 35.3;
      O     DB23.DBX 35.3;
      O     DB24.DBX 35.3;
      );
      O;
      A     "MSTT_1".B_Chan1Start;
      A     DB21.DBX 35.3;
      O;
      A     "MSTT_1".B_Chan2Start;
      A     DB22.DBX 35.3;
      O;
      A     "MSTT_2".B_Chan3Start;
      A     DB23.DBX 35.3;
      O;
      A     "MSTT_2".B_Chan4Start;
      A     DB24.DBX 35.3;
      O     "MSTT_1".B_Reset;
      R     "ПриостПл";
NETWORK
TITLE = Velocity/spindle speed limitation
      O     "РежТолчПл";
      O;
      AN    "ОгрПоднято";
      AN    "On";
      =     DB31.DBX 3.6;
NETWORK
TITLE = Feed stop/spindle stop
      AN    "ЗагЗажата";
      AN    "РежТолчПл";
      AN    "РежПереклПл";
      O     "ПриостПл";
      =     DB31.DBX 4.3;
NETWORK
TITLE = Delete distance to go/Spindel-Reset
      AN    "РазрПл";
      A     "ТОстПл";
      O     "MSTT_1".B_Reset;
      =     DB31.DBX 2.2;
NETWORK
TITLE = Управление смазкой планшайбы
      CALL  "Table_Lub";
      NOP   0;
NETWORK
TITLE = Скорость планшайбы Nact < N min
      A     DB31.DBX 61.4;
      =     "СкорПл0";
NETWORK
TITLE = Двигатель главного привода и планшайба не вращаются
      A     "АвтВентГП";
      A     "СкорПл0";
      =     "НетДвижГП";
NETWORK
TITLE = Планшайба стоит
      AN    "ПускПл";
      A     "НетДвижГП";
      =     "ГПСтоит";
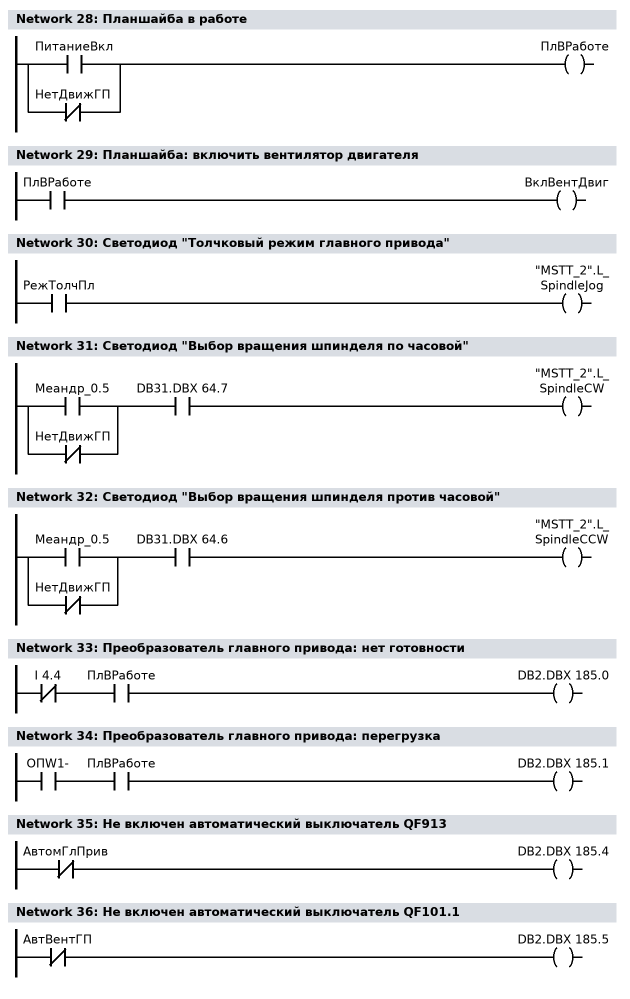
NETWORK
TITLE = Планшайба в работе
      O     "ПитаниеВкл";
      ON    "НетДвижГП";
      =     "ПлВРаботе";
NETWORK
TITLE = Планшайба: включить вентилятор двигателя
      A     "ПлВРаботе";
      =     "ВклВентДвиг";
NETWORK
TITLE = Светодиод "Толчковый режим главного привода"
      A     "РежТолчПл";
      =     "MSTT_2".L_SpindleJog;
NETWORK
TITLE = Светодиод "Выбор вращения шпинделя по часовой"
      A(;
      O     "Меандр_0.5";
      ON    "НетДвижГП";
      );
      A     DB31.DBX 64.7;
      =     "MSTT_2".L_SpindleCW;
NETWORK
TITLE = Светодиод "Выбор вращения шпинделя против часовой"
      A(;
      O     "Меандр_0.5";
      ON    "НетДвижГП";
      );
      A     DB31.DBX 64.6;
      =     "MSTT_2".L_SpindleCCW;
NETWORK
TITLE = Преобразователь главного привода: нет готовности
      AN    I 4.4;
      A     "ПлВРаботе";
      =     DB2.DBX 185.0;
NETWORK
TITLE = Преобразователь главного привода: перегрузка
      A     "ОПW1-";
      A     "ПлВРаботе";
      =     DB2.DBX 185.1;
NETWORK
TITLE = Не включен автоматический выключатель QF913
      AN    "АвтомГлПрив";
      =     DB2.DBX 185.4;
NETWORK
TITLE = Не включен автоматический выключатель QF101.1
      AN    "АвтВентГП";
      =     DB2.DBX 185.5;
END_FUNCTION_BLOCK

// FC 2: know-how protected block, not included

// FC 3: know-how protected block, not included

// FC 5: know-how protected block, not included

// FC 6: know-how protected block, not included

// FC 7: know-how protected block, not included

// FC 8: know-how protected block, not included

// FC 9: know-how protected block, not included

// FC 10: know-how protected block, not included

FUNCTION FC 12 : VOID
AUTHOR : NUMERIK
FAMILY : _800D
NAME : Basics
VERSION : 2.7
VAR_INPUT
  Chan : BYTE ;	//Index of Chan
END_VAR
BEGIN
NETWORK
TITLE =
END_FUNCTION

// FC 13: know-how protected block, not included

// FC 16: know-how protected block, not included

// FC 17: know-how protected block, not included

// FC 18: know-how protected block, not included

// FC 19: know-how protected block, not included

// FC 20: know-how protected block, not included

// FC 21: know-how protected block, not included

// FC 22: know-how protected block, not included

// FC 24: know-how protected block, not included

// FC 25: know-how protected block, not included

// FC 26: know-how protected block, not included

FUNCTION "PowerOn" : VOID	// FC 100
AUTHOR : SEDIN
VERSION : 0.1
VAR_TEMP
  NoMotion : BOOL ;	//Органы станка неподвижны
END_VAR
BEGIN
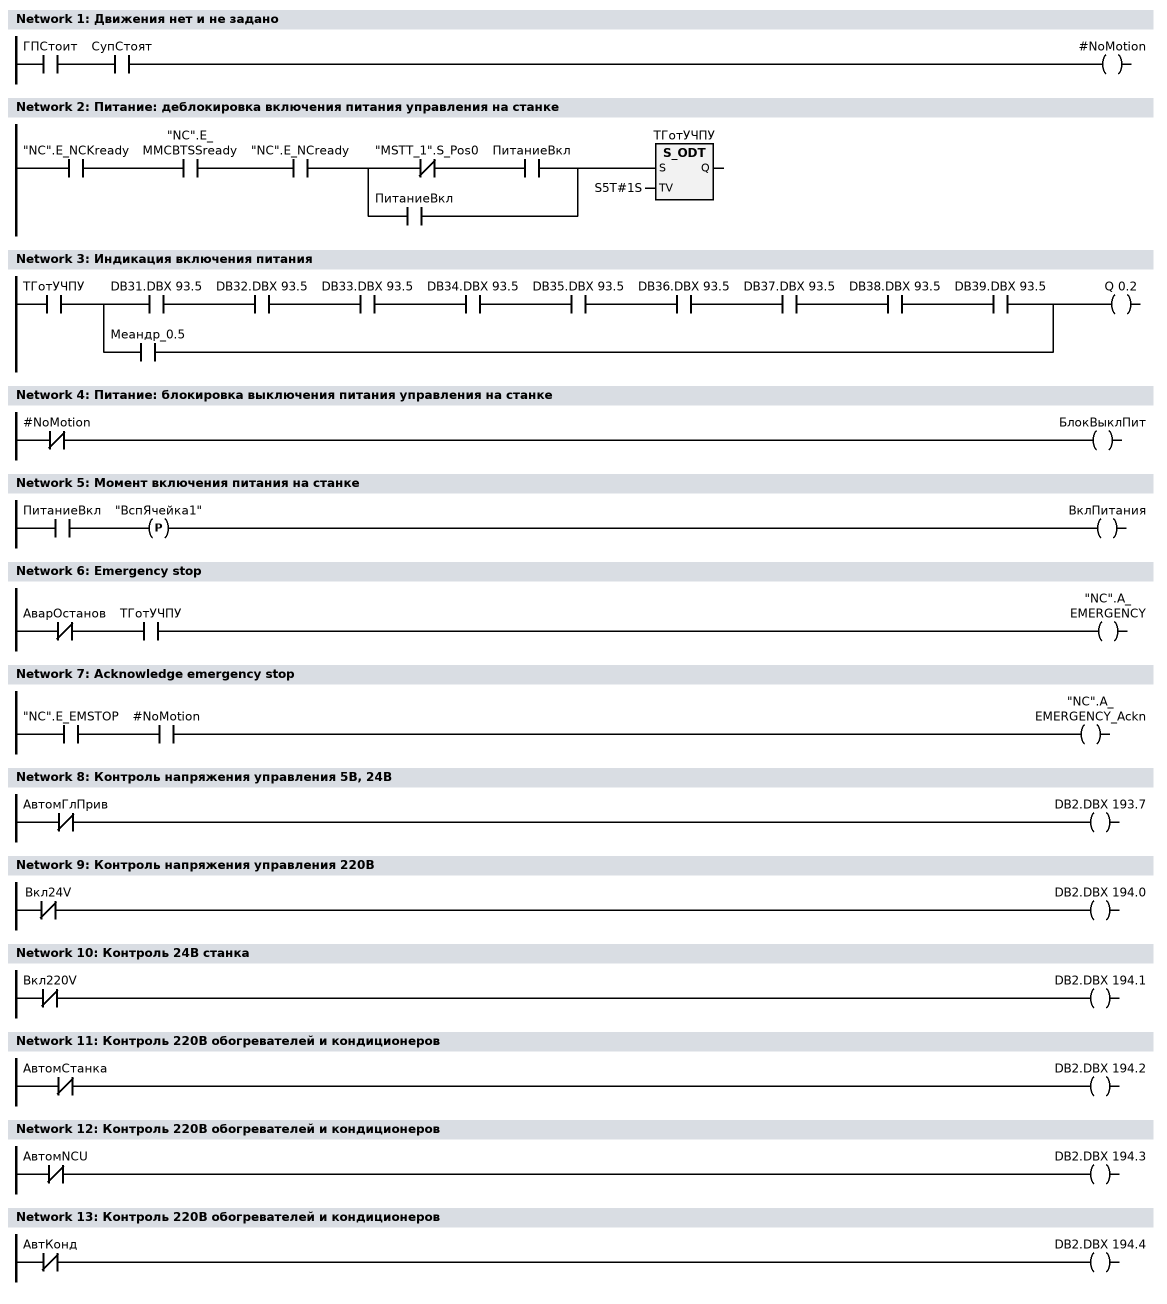
NETWORK
TITLE = Движения нет и не задано
      A     "ГПСтоит";
      A     "СупСтоят";
      =     #NoMotion;
NETWORK
TITLE = Питание: деблокировка включения питания управления на станке
      A     "NC".E_NCKready;
      A     "NC".E_MMCBTSSready;
      A     "NC".E_NCready;
      A(;
      AN    "MSTT_1".S_Pos0;
      A     "ПитаниеВкл";
      O     "ПитаниеВкл";
      );
      L     S5T#1S;
      SD    "ТГотУЧПУ";
      NOP   0;
      NOP   0;
      NOP   0;
      NOP   0;
NETWORK
TITLE = Индикация включения питания
      A     "ТГотУЧПУ";
      A(;
      A     DB31.DBX 93.5;
      A     DB32.DBX 93.5;
      A     DB33.DBX 93.5;
      A     DB34.DBX 93.5;
      A     DB35.DBX 93.5;
      A     DB36.DBX 93.5;
      A     DB37.DBX 93.5;
      A     DB38.DBX 93.5;
      A     DB39.DBX 93.5;
      O     "Меандр_0.5";
      );
      =     Q 0.2;
NETWORK
TITLE = Питание: блокировка выключения питания управления на станке
      AN    #NoMotion;
      =     "БлокВыклПит";
NETWORK
TITLE = Момент включения питания на станке
      A     "ПитаниеВкл";
      BLD   100;
      FP    "ВспЯчейка1";
      =     "ВклПитания";
NETWORK
TITLE = Emergency stop                        
      AN    "АварОстанов";
      A     "ТГотУЧПУ";
      =     "NC".A_EMERGENCY;
NETWORK
TITLE = Acknowledge emergency stop                      
      A     "NC".E_EMSTOP;
      A     #NoMotion;
      =     "NC".A_EMERGENCY_Ackn;
NETWORK
TITLE = Контроль напряжения управления 5В, 24В
      AN    "АвтомГлПрив";
      =     DB2.DBX 193.7;
NETWORK
TITLE = Контроль напряжения управления 220В
      AN    "Вкл24V";
      =     DB2.DBX 194.0;
NETWORK
TITLE = Контроль 24В станка
      AN    "Вкл220V";
      =     DB2.DBX 194.1;
NETWORK
TITLE = Контроль 220В обогревателей и кондиционеров
      AN    "АвтомСтанка";
      =     DB2.DBX 194.2;
NETWORK
TITLE = Контроль 220В обогревателей и кондиционеров
      AN    "АвтомNCU";
      =     DB2.DBX 194.3;
NETWORK
TITLE = Контроль 220В обогревателей и кондиционеров
      AN    "АвтКонд";
      =     DB2.DBX 194.4;
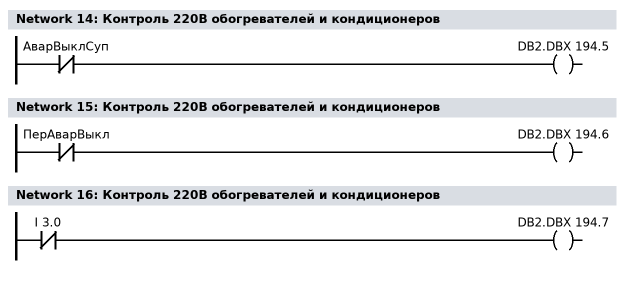
NETWORK
TITLE = Контроль 220В обогревателей и кондиционеров
      AN    "АварВыклСуп";
      =     DB2.DBX 194.5;
NETWORK
TITLE = Контроль 220В обогревателей и кондиционеров
      AN    "ПерАварВыкл";
      =     DB2.DBX 194.6;
NETWORK
TITLE = Контроль 220В обогревателей и кондиционеров
      AN    I 3.0;
      =     DB2.DBX 194.7;
END_FUNCTION

FUNCTION "Infeed_Module" : VOID	// FC 101
AUTHOR : SEDIN
VERSION : 0.1
VAR_TEMP
  Aux : ARRAY  [1 .. 10 ] OF BOOL ;
END_VAR
BEGIN
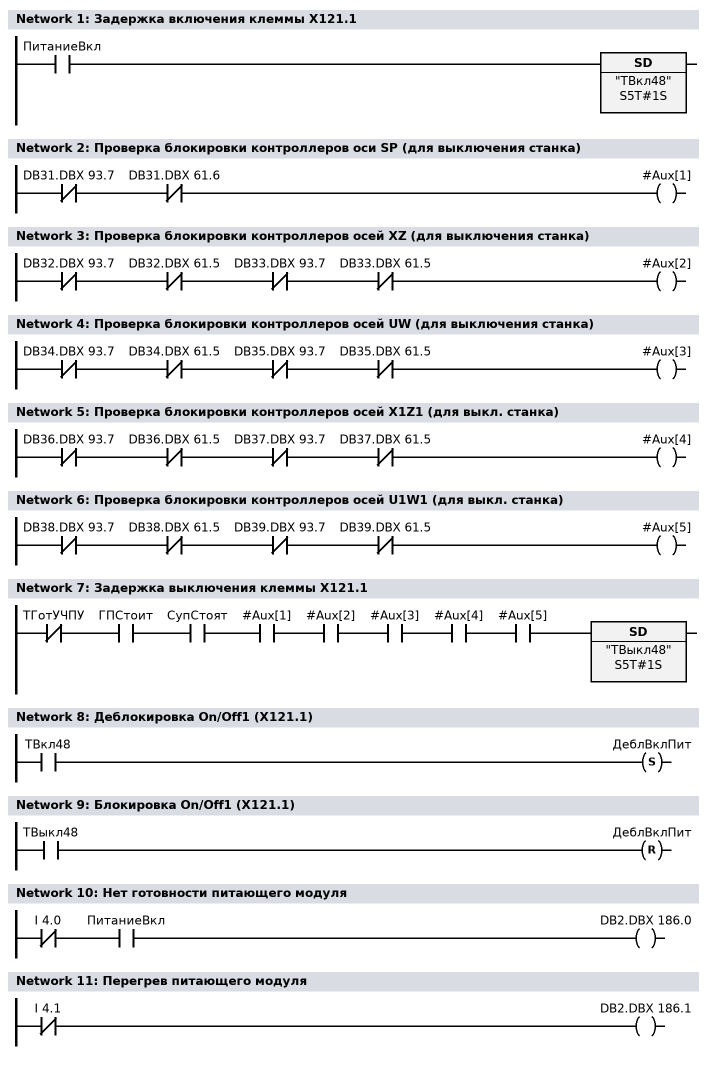
NETWORK
TITLE = Задержка включения клеммы X121.1
      A     "ПитаниеВкл";
      L     S5T#1S;
      SD    "ТВкл48";
NETWORK
TITLE = Проверка блокировки контроллеров оси SP (для выключения станка)
      AN    DB31.DBX 93.7;
      AN    DB31.DBX 61.6;
      =     #Aux[1];
NETWORK
TITLE = Проверка блокировки контроллеров осей XZ (для выключения станка)
      AN    DB32.DBX 93.7;
      AN    DB32.DBX 61.5;
      AN    DB33.DBX 93.7;
      AN    DB33.DBX 61.5;
      =     #Aux[2];
NETWORK
TITLE = Проверка блокировки контроллеров осей UW (для выключения станка)
      AN    DB34.DBX 93.7;
      AN    DB34.DBX 61.5;
      AN    DB35.DBX 93.7;
      AN    DB35.DBX 61.5;
      =     #Aux[3];
NETWORK
TITLE = Проверка блокировки контроллеров осей X1Z1 (для выкл. станка)
      AN    DB36.DBX 93.7;
      AN    DB36.DBX 61.5;
      AN    DB37.DBX 93.7;
      AN    DB37.DBX 61.5;
      =     #Aux[4];
NETWORK
TITLE = Проверка блокировки контроллеров осей U1W1 (для выкл. станка)
      AN    DB38.DBX 93.7;
      AN    DB38.DBX 61.5;
      AN    DB39.DBX 93.7;
      AN    DB39.DBX 61.5;
      =     #Aux[5];
NETWORK
TITLE = Задержка выключения клеммы X121.1
      AN    "ТГотУЧПУ";
      A     "ГПСтоит";
      A     "СупСтоят";
      A     #Aux[1];
      A     #Aux[2];
      A     #Aux[3];
      A     #Aux[4];
      A     #Aux[5];
      L     S5T#1S;
      SD    "ТВыкл48";
NETWORK
TITLE = Деблокировка On/Off1 (X121.1)
      A     "ТВкл48";
      S     "ДеблВклПит";
NETWORK
TITLE = Блокировка On/Off1 (X121.1)
      A     "ТВыкл48";
      R     "ДеблВклПит";
NETWORK
TITLE = Нет готовности питающего модуля
      AN    I 4.0;
      A     "ПитаниеВкл";
      =     DB2.DBX 186.0;
NETWORK
TITLE = Перегрев питающего модуля
      AN    I 4.1;
      =     DB2.DBX 186.1;
END_FUNCTION

FUNCTION "Aux_Function" : VOID	// FC 107
AUTHOR : SEDIN
VERSION : 0.1
VAR_TEMP
  Count : INT ;	//Счетчик
END_VAR
BEGIN
NETWORK
TITLE = Открытие блока данных 1 канала и блока вспомогательных функций
      OPN   "Chan1";
      LAR1  P#194.0;
      OPN   DI 130;
      LAR2  P#0.0;
NETWORK
TITLE = Передача данных о вспомогательных функциях канала 1
      L     39;
L001: L     DBW [AR1,P#0.0];
      T     DIW [AR2,P#0.0];
      +AR1  P#2.0;
      +AR2  P#2.0;
      TAK;
      LOOP  L001;
NETWORK
TITLE = Открытие блока данных 2 канала и блока вспомогательных функций
      OPN   "Chan2";
      LAR1  P#194.0;
      OPN   DI 130;
      LAR2  P#0.0;
NETWORK
TITLE = Передача данных о вспомогательных функциях канала 2
      L     39;
L002: T     #Count;
      L     DBW [AR1,P#0.0];
      L     DIW [AR2,P#0.0];
      OW;
      T     DIW [AR2,P#0.0];
      +AR1  P#2.0;
      +AR2  P#2.0;
      L     #Count;
      LOOP  L002;
NETWORK
TITLE = Открытие блока данных 3 канала и блока вспомогательных функций
      OPN   "Chan3";
      LAR1  P#194.0;
      OPN   DI 130;
      LAR2  P#0.0;
NETWORK
TITLE = Передача данных о вспомогательных функциях канала 3
      L     39;
L003: T     #Count;
      L     DBW [AR1,P#0.0];
      L     DIW [AR2,P#0.0];
      OW;
      T     DIW [AR2,P#0.0];
      +AR1  P#2.0;
      +AR2  P#2.0;
      L     #Count;
      LOOP  L003;
NETWORK
TITLE = Открытие блока данных 4 канала и блока вспомогательных функций
      OPN   "Chan4";
      LAR1  P#194.0;
      OPN   DI 130;
      LAR2  P#0.0;
NETWORK
TITLE = Передача данных о вспомогательных функциях канала 4
      L     39;
L004: T     #Count;
      L     DBW [AR1,P#0.0];
      L     DIW [AR2,P#0.0];
      OW;
      T     DIW [AR2,P#0.0];
      +AR1  P#2.0;
      +AR2  P#2.0;
      L     #Count;
      LOOP  L004;
END_FUNCTION

FUNCTION "Correction" : VOID	// FC 108
AUTHOR : SEDIN
VERSION : 0.1
VAR_TEMP
  OverrideSp : WORD ;	//Корректор шпинделя
  OverrideF1 : WORD ;	//Корректор подачи суппорта 1
  OverrideF2 : WORD ;	//Корректор подачи суппорта 2
  OverrideF3 : WORD ;	//Корректор подачи суппорта 3
  OverrideF4 : WORD ;	//Корректор подачи суппорта 4
  OverHHU : WORD ;	//Корректор подачи от HHU
  Temp1 : WORD ;
  Temp2 : INT ;
  Temp3 : INT ;
  B_Continuous : BOOL ;	//Отключение инкриментальных перемещений от ВП
  Pos_INC1 : BOOL ;
  Pos_INC10 : BOOL ;
  Pos_INC100 : BOOL ;
END_VAR
BEGIN
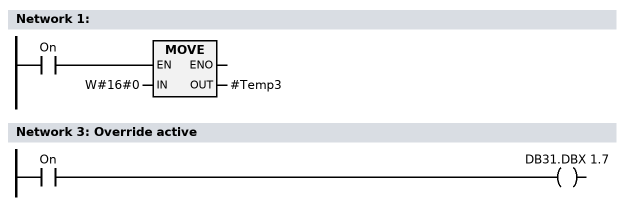
NETWORK
TITLE =
      A     "On";
      JNB   _001;
      L     W#16#0;
      T     #Temp3;
_001: NOP   0;
NETWORK
TITLE = Корректор шпинделя
      A     "On";
      =     L 19.0;
      A     L 19.0;
      A     "КоррПлБит0";
      =     L 17.0;
      A     L 19.0;
      A     "КоррПлБит1";
      =     L 17.1;
      A     L 19.0;
      A     "КоррПлБит2";
      =     L 17.2;
      A     L 19.0;
      A     "КоррПлБит3";
      =     L 17.3;
      A     L 19.0;
      A     "КоррПлБит4";
      =     L 17.4;
NETWORK
TITLE = Override active
      A     "On";
      =     DB31.DBX 1.7;
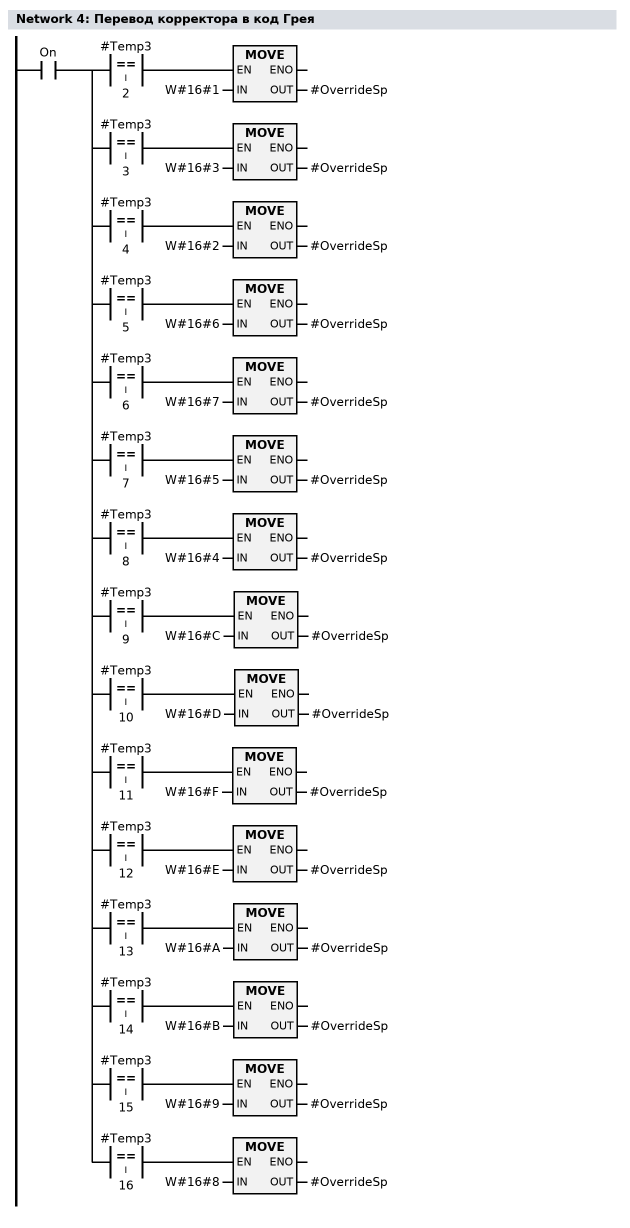
NETWORK
TITLE = Перевод корректора в код Грея
      A     "On";
      =     L 19.0;
      A     L 19.0;
      A(;
      L     #Temp3;
      L     2;
      ==I;
      );
      JNB   _002;
      L     W#16#1;
      T     #OverrideSp;
_002: NOP   0;
      A     L 19.0;
      A(;
      L     #Temp3;
      L     3;
      ==I;
      );
      JNB   _003;
      L     W#16#3;
      T     #OverrideSp;
_003: NOP   0;
      A     L 19.0;
      A(;
      L     #Temp3;
      L     4;
      ==I;
      );
      JNB   _004;
      L     W#16#2;
      T     #OverrideSp;
_004: NOP   0;
      A     L 19.0;
      A(;
      L     #Temp3;
      L     5;
      ==I;
      );
      JNB   _005;
      L     W#16#6;
      T     #OverrideSp;
_005: NOP   0;
      A     L 19.0;
      A(;
      L     #Temp3;
      L     6;
      ==I;
      );
      JNB   _006;
      L     W#16#7;
      T     #OverrideSp;
_006: NOP   0;
      A     L 19.0;
      A(;
      L     #Temp3;
      L     7;
      ==I;
      );
      JNB   _007;
      L     W#16#5;
      T     #OverrideSp;
_007: NOP   0;
      A     L 19.0;
      A(;
      L     #Temp3;
      L     8;
      ==I;
      );
      JNB   _008;
      L     W#16#4;
      T     #OverrideSp;
_008: NOP   0;
      A     L 19.0;
      A(;
      L     #Temp3;
      L     9;
      ==I;
      );
      JNB   _009;
      L     W#16#C;
      T     #OverrideSp;
_009: NOP   0;
      A     L 19.0;
      A(;
      L     #Temp3;
      L     10;
      ==I;
      );
      JNB   _00a;
      L     W#16#D;
      T     #OverrideSp;
_00a: NOP   0;
      A     L 19.0;
      A(;
      L     #Temp3;
      L     11;
      ==I;
      );
      JNB   _00b;
      L     W#16#F;
      T     #OverrideSp;
_00b: NOP   0;
      A     L 19.0;
      A(;
      L     #Temp3;
      L     12;
      ==I;
      );
      JNB   _00c;
      L     W#16#E;
      T     #OverrideSp;
_00c: NOP   0;
      A     L 19.0;
      A(;
      L     #Temp3;
      L     13;
      ==I;
      );
      JNB   _00d;
      L     W#16#A;
      T     #OverrideSp;
_00d: NOP   0;
      A     L 19.0;
      A(;
      L     #Temp3;
      L     14;
      ==I;
      );
      JNB   _00e;
      L     W#16#B;
      T     #OverrideSp;
_00e: NOP   0;
      A     L 19.0;
      A(;
      L     #Temp3;
      L     15;
      ==I;
      );
      JNB   _00f;
      L     W#16#9;
      T     #OverrideSp;
_00f: NOP   0;
      A     L 19.0;
      A(;
      L     #Temp3;
      L     16;
      ==I;
      );
      JNB   _010;
      L     W#16#8;
      T     #OverrideSp;
_010: NOP   0;
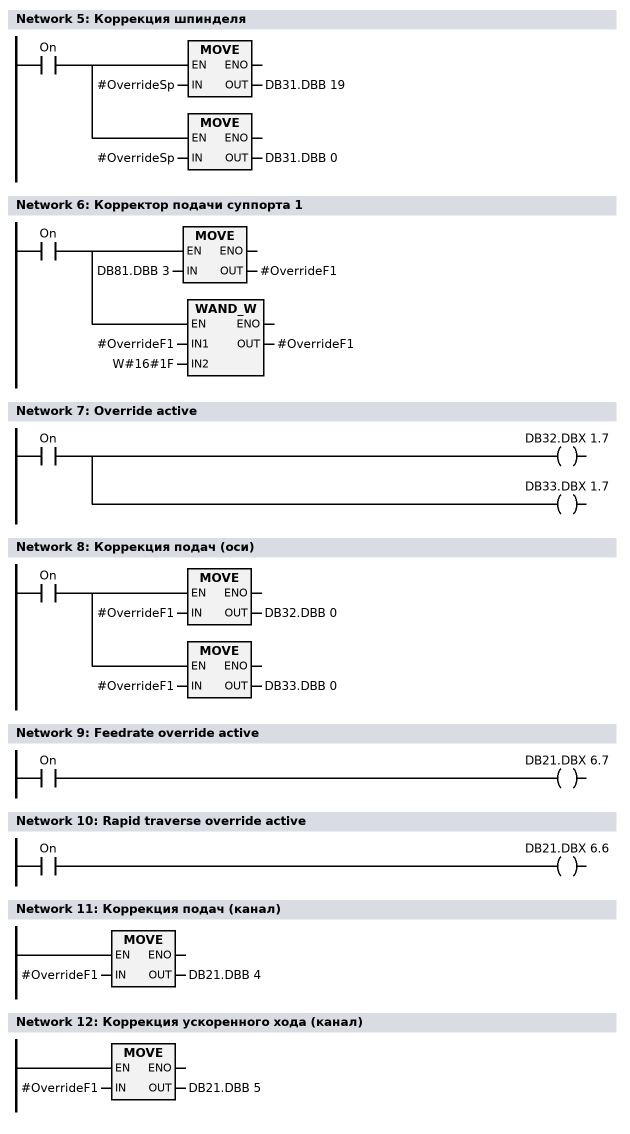
NETWORK
TITLE = Коррекция шпинделя
      A     "On";
      =     L 19.0;
      A     L 19.0;
      JNB   _011;
      L     #OverrideSp;
      T     DB31.DBB 19;
_011: NOP   0;
      A     L 19.0;
      JNB   _012;
      L     #OverrideSp;
      T     DB31.DBB 0;
_012: NOP   0;
NETWORK
TITLE = Корректор подачи суппорта 1
      A     "On";
      =     L 19.0;
      A     L 19.0;
      JNB   _013;
      L     DB81.DBB 3;
      T     #OverrideF1;
_013: NOP   0;
      A     L 19.0;
      JNB   _014;
      L     #OverrideF1;
      L     W#16#1F;
      AW;
      T     #OverrideF1;
_014: NOP   0;
NETWORK
TITLE = Override active
      A     "On";
      =     DB32.DBX 1.7;
      =     DB33.DBX 1.7;
NETWORK
TITLE = Коррекция подач (оси)
      A     "On";
      =     L 19.0;
      A     L 19.0;
      JNB   _015;
      L     #OverrideF1;
      T     DB32.DBB 0;
_015: NOP   0;
      A     L 19.0;
      JNB   _016;
      L     #OverrideF1;
      T     DB33.DBB 0;
_016: NOP   0;
NETWORK
TITLE = Feedrate override active
      A     "On";
      =     DB21.DBX 6.7;
NETWORK
TITLE = Rapid traverse override active
      A     "On";
      =     DB21.DBX 6.6;
NETWORK
TITLE = Коррекция подач (канал)
      L     #OverrideF1;
      T     DB21.DBB 4;
      NOP   0;
NETWORK
TITLE = Коррекция ускоренного хода (канал)
      L     #OverrideF1;
      T     DB21.DBB 5;
      NOP   0;
NETWORK
TITLE = Корректор подачи суппорта 2
      A     "On";
      =     L 19.0;
      A     L 19.0;
      JNB   _017;
      L     DB81.DBB 0;
      T     #Temp1;
_017: NOP   0;
      A     L 19.0;
      JNB   _018;
      L     #Temp1;
      L     W#16#F0;
      AW;
      T     #Temp1;
_018: NOP   0;
      A     L 19.0;
      JNB   _019;
      L     W#16#4;
      L     #Temp1;
      SRW;
      T     #Temp1;
_019: NOP   0;
      A     L 19.0;
      JNB   _01a;
      L     #Temp1;
      T     #Temp2;
_01a: NOP   0;
